  gripCyl.homeSensor[0]:= HomeSensor_gripCyl ;
  gripCyl.workSensor[0]:= WorkSensor_gripCyl ;
  HomeValve_gripCyl:= gripCyl.homeValve ;
  WorkValve_gripCyl:= gripCyl.workValve ;
  gripCyl.homeSensorLabel[0] := HomeLabel_gripCyl;
  gripCyl.workSensorLabel[0] := WorkLabel_gripCyl;
  
  jackCyl.homeSensor[0]:= HomeSensor_jackCyl ;
  jackCyl.workSensor[0]:= WorkSensor_jackCyl ;
  HomeValve_jackCyl:= jackCyl.homeValve ;
  WorkValve_jackCyl:= jackCyl.workValve ;
  jackCyl.homeSensorLabel[0] := HomeLabel_jackCyl;
  jackCyl.workSensorLabel[0] := WorkLabel_jackCyl;
  
  HomeValve_blow:= blow.homeValve ;
  WorkValve_blow:= blow.workValve ;
  
  fixCyl.homeSensor[0]:= HomeSensor_fixCyl ;
  fixCyl.workSensor[0]:= WorkSensor_fixCyl ;
  HomeValve_fixCyl:= fixCyl.homeValve ;
  WorkValve_fixCyl:= fixCyl.workValve ;
  fixCyl.homeSensorLabel[0] := HomeLabel_fixCyl;
  fixCyl.workSensorLabel[0] := WorkLabel_fixCyl;
  
  stepFixCyl.homeSensor[0]:= HomeSensor_stepFixCyl ;
  stepFixCyl.workSensor[0]:= WorkSensor_stepFixCyl ;
  HomeValve_stepFixCyl:= stepFixCyl.homeValve ;
  WorkValve_stepFixCyl:= stepFixCyl.workValve ;
  stepFixCyl.homeSensorLabel[0] := HomeLabel_stepFixCyl;
  stepFixCyl.workSensorLabel[0] := WorkLabel_stepFixCyl;
  
// Parameter 

  JacketStrippingData.Blow.homeSensorDisabled[0] := TRUE;
  JacketStrippingData.Blow.workSensorDisabled[0] := TRUE;
  
  rotateAxis.modulo.divisor := 2;
  rotateAxis.modulo.stepPoint :=1;
  rotateAxis.modulo.factor :=360;
  rotateAxis.modulo.mode := 1;
  rotateAxis.modulo.enable :=TRUE;
  rotateAxis.posUnit			:='deg';
  rotateAxis.veloUnit			:='deg/s';
  rotateAxis.accDecUnit	  :="deg/s²";
  
  cutAxis.movePosNum := 18;
  transferAxis.movePosNum := 15;
  rotateAxis.velocity :=1000;
  
  rotateAxis.Override := JacketStrippingData.CPP.override;
  TransferAxis.Override := JacketStrippingData.CPP.override;
  CutAxis.Override := JacketStrippingData.CPP.override;
  
  tonOn(IN:= onePlus, PT:= T#2S, Q=> , ET=> );
  tonOff(IN:= NOT onePlus, PT:= T#2S, Q=> , ET=> );
  IF tonOn.Q OR tonOff.Q THEN
    onePlus := NOT onePlus;
  END_IF
  
  mcWriteParameterPersistent(
    Axis:= rotateAxis.axis, 
    Execute:= onePlus, 
    ParameterNumber:= 1045, 
    Value:= 360.0, 
    Done=> , 
    Busy=> , 
    Error=> , 
    ErrorID=> );
    


//DATA 模拟

  IF NOT activated THEN
  
  activated:=TRUE;
  
  JacketStripping.Imm.Machine_airOn := TRUE;
  JacketStripping.Imm.Machine_allDoorClosed:= TRUE;
  JacketStripping.Imm.Machine_eStop:= TRUE;
  JacketStripping.Imm.Machine_safety:= TRUE;
  JacketStripping.Imm.Machine_manualMode:= TRUE;
  
  JacketStripping.Imm.carrierInPos := TRUE;
  JacketStripping.Imm.carrierPos := ENUM_CarrierPos.Left;
  JacketStripping.Imm.StationCanRun := TRUE;
  JacketStrippingData.CPP.override := 100;
  
  JacketStrippingData.CutAxis.movePos[HOME_CUT] := 40;
  JacketStrippingData.CutAxis.movePos[FIRST_PRECUT_CUT] := 30;
  JacketStrippingData.CutAxis.movePos[FIRST_CUT_CUT] := 10;
  JacketStrippingData.CutAxis.movePos[FIRST_BACK_CUT] := 20;
  JacketStrippingData.CutAxis.movePos[SECOND_PRECUT_CUT] := 25;
  JacketStrippingData.CutAxis.movePos[SECOND_CUT_CUT] :=5;
  JacketStrippingData.CutAxis.movePos[SECOND_BACK_CUT] := 15;
  
  JacketStrippingData.TransferAxis.movePos[HOME_TRANS] := 0;
  JacketStrippingData.TransferAxis.movePos[FIRST_CUT_TRANS] := 200;
  JacketStrippingData.TransferAxis.movePos[FIRST_BACK_TRANS] := 50;
  JacketStrippingData.TransferAxis.movePos[SECOND_CUT_TRANS] := 100;
  JacketStrippingData.TransferAxis.movePos[SECOND_BACK_TRANS] := 25;
  
  JacketStrippingData.GripCyl.homeSensorDisabled[0] := TRUE;
  JacketStrippingData.GripCyl.workSensorDisabled[0] := TRUE;
  JacketStrippingData.JackCyl.homeSensorDisabled[0] := TRUE;
  JacketStrippingData.JackCyl.workSensorDisabled[0] := TRUE;
  JacketStrippingData.FixCyl.homeSensorDisabled[0] := TRUE;
  JacketStrippingData.FixCyl.workSensorDisabled[0] := TRUE;
  JacketStrippingData.StepFixCyl.homeSensorDisabled[0] := TRUE;
  JacketStrippingData.StepFixCyl.workSensorDisabled[0] := TRUE;
  JacketStrippingData.GripCyl.homeTime := 500;
  JacketStrippingData.GripCyl.workTime := 500;
  JacketStrippingData.JackCyl.homeTime := 500;
  JacketStrippingData.JackCyl.workTime := 500;
  JacketStrippingData.FixCyl.homeTime := 500;
  JacketStrippingData.FixCyl.workTime := 500;
  JacketStrippingData.StepFixCyl.homeTime := 500;
  JacketStrippingData.StepFixCyl.workTime := 500;
  JacketStrippingData.Blow.homeTime := 500;
  JacketStrippingData.Blow.workTime := 500;
  
  END_IF
END_ACTION

ACTION StepAuto:
IF NOT station.initDone THEN
	station.flow[AUTO].actStep:=0;
ELSIF station.running 
THEN

CASE station.flow[AUTO].actStep OF

//	Home Step
0:
IF station.disabled
	AND station.canRun
  AND JacketStripping.Imm.allObjectInitPos
  AND NOT machine.stopping
  AND NOT station.cycleRunning
THEN
	JacketStripping.Imm.stationDone:=TRUE;
END_IF

IF (station.cycleRunning
		OR station.canRun
      AND JacketStripping.Imm.allObjectInitPos
			AND NOT station.Done
			AND NOT station.Disabled
      AND NOT machine.stopping
	)
	AND JacketStripping.Imm.carrierInPos
THEN
	station.flow[AUTO].actStep:=10;
	station.cycleTimeStart:=TRUE;
	station.cycleTimeEnd:=FALSE;
END_IF


//	fixCyl up
10:
IF JacketStripping.Imm.carrierPos= ENUM_CarrierPos.Left THEN
  fixCyl.auto:= TRUE;
  JacketStripping.Imm.carrierLeftProductState := 0;
	IF fixCyl.inWork THEN
		station.flow[AUTO].actStep:=station.flow[AUTO].actStep + 10;
	END_IF
ELSIF JacketStripping.Imm.carrierPos= ENUM_CarrierPos.Right THEN
  stepFixCyl.auto:= TRUE;
  JacketStripping.Imm.carrierRightProductState := 0;
	IF stepFixCyl.inWork THEN
		station.flow[AUTO].actStep:=station.flow[AUTO].actStep + 10;
	END_IF
END_IF


//	jackCyl up
20:
jackCyl.auto:=TRUE;
IF jackCyl.inWork THEN
	station.flow[AUTO].actStep:=station.flow[AUTO].actStep + 10;
END_IF

//	gripCyl close
30:
gripCyl.auto:=TRUE;
IF gripCyl.inWork THEN
	station.flow[AUTO].actStep:=station.flow[AUTO].actStep + 10;
END_IF

//transferAxis to firstCut pos
40:
transferAxis.moveAutoNo:=FIRST_CUT_TRANS;
IF transferAxis.inPos[FIRST_CUT_TRANS] THEN 
	station.flow[AUTO].actStep:=station.flow[AUTO].actStep + 10;
END_IF


//cutAxis to firstPreCut pos
50:
cutAxis.moveAutoNo:=FIRST_PRECUT_CUT;
rotateAxis.velocityAuto:=TRUE;
IF cutAxis.inPos[FIRST_PRECUT_CUT] THEN 
	station.flow[AUTO].actStep:=station.flow[AUTO].actStep + 10;
END_IF


//rotateAxis start
60:
IF rotateAxis.InVelocity THEN 
	station.flow[AUTO].actStep:=station.flow[AUTO].actStep + 10;
END_IF


//cutAxis to firstCut pos
70:
cutAxis.moveAutoNo:= FIRST_CUT_CUT;
IF cutAxis.inPos[FIRST_CUT_CUT] THEN 
	station.flow[AUTO].actStep:=station.flow[AUTO].actStep + 10;
END_IF
firstCutTimer(IN:=FALSE,PT:=UDINT_TO_TIME(JacketStrippingData.CPP.FirstCutTime),Q=>,ET=>);


//Wait firstCut delay
80:
firstCutTimer(IN:=TRUE,PT:=UDINT_TO_TIME(JacketStrippingData.CPP.FirstCutTime),Q=>,ET=>);
IF firstCutTimer.Q THEN
	station.flow[AUTO].actStep:=station.flow[AUTO].actStep + 10;
END_IF


//rotateAxis end
90:
  rotateAxis.stopAuto:=TRUE;
  IF rotateAxis.Axis.Status.NotMoving THEN
    rotateAxis.stopAuto:=FALSE;
    station.flow[AUTO].actStep:=station.flow[AUTO].actStep + 5;
	END_IF
  
//cutAxis to firstBack pos  
95:
  rotateAxis.stopAuto:=FALSE;
cutAxis.moveAutoNo:= FIRST_BACK_CUT;
IF cutAxis.inPos[FIRST_BACK_CUT] THEN 	
	station.flow[AUTO].actStep:=station.flow[AUTO].actStep + 5;
END_IF
firstOpenTimer(IN:=FALSE,PT:= UDINT_TO_TIME(JacketStrippingData.CPP.firstOpenTime),Q=>,ET=>);


//Wait firstOpen delay
100:
firstOpenTimer(IN:=TRUE,PT:=UDINT_TO_TIME(JacketStrippingData.CPP.firstOpenTime),Q=>,ET=>);
IF firstOpenTimer.Q THEN
	station.flow[AUTO].actStep:=station.flow[AUTO].actStep + 10;
END_IF

110:
//transferAxis to firstBack pos
transferAxis.moveAutoNo:=FIRST_BACK_TRANS;
IF transferAxis.inPos[FIRST_BACK_TRANS] THEN
	IF NOT JacketStrippingData.CPP.secondCutEnable THEN
		IF JacketStripping.Imm.carrierPos = ENUM_CarrierPos.Left THEN
			JacketStripping.Imm.carrierLeftProductState:=ENUM_ProductState.Good;
		ELSIF JacketStripping.Imm.carrierPos =ENUM_CarrierPos.Right THEN
			JacketStripping.Imm.carrierRightProductState:=ENUM_ProductState.Good;
		END_IF
		station.flow[AUTO].actStep:=900;
	ELSE
		station.flow[AUTO].actStep:=station.flow[AUTO].actStep + 10;
	END_IF
END_IF


//cutAxis to home pos
120:
cutAxis.moveAutoNo:= HOME_CUT;
IF cutAxis.inPos[HOME_CUT] THEN 
	station.flow[AUTO].actStep:=station.flow[AUTO].actStep + 80;
END_IF

//transferAxis to secondCut pos
200:
transferAxis.moveAutoNo:=SECOND_CUT_TRANS;
IF transferAxis.inPos[SECOND_CUT_TRANS] THEN
  	station.flow[AUTO].actStep:=station.flow[AUTO].actStep + 10;
END_IF


//cutAxis to secondPreCut pos
210:
rotateAxis.VelocityAuto:=TRUE;
cutAxis.moveAutoNo:= SECOND_PRECUT_CUT;
IF cutAxis.inPos[SECOND_PRECUT_CUT] THEN 
	station.flow[AUTO].actStep:=station.flow[AUTO].actStep + 10;
END_IF


//rotateAxis start
220:
IF rotateAxis.InVelocity THEN 
	station.flow[AUTO].actStep:=station.flow[AUTO].actStep + 10;
END_IF


//cutAxis to secondCut pos
230:

cutAxis.moveAutoNo:= SECOND_CUT_CUT;
IF cutAxis.inPos[SECOND_CUT_CUT] THEN 
	station.flow[AUTO].actStep:=station.flow[AUTO].actStep + 10;
END_IF
SecondCutTimer(IN:=FALSE,PT:=UDINT_TO_TIME(JacketStrippingData.CPP.SecondCutTime),Q=>,ET=>);


//Wait secondCut delay
240:
SecondCutTimer(IN:=TRUE,PT:=UDINT_TO_TIME(JacketStrippingData.CPP.SecondCutTime),Q=>,ET=>);
IF SecondCutTimer.Q THEN
	station.flow[AUTO].actStep:=station.flow[AUTO].actStep + 10;
END_IF

//rotateAxis end
250:
  rotateAxis.stopAuto:=TRUE;
  IF rotateAxis.Axis.Status.NotMoving THEN
    rotateAxis.stopAuto:=FALSE;
    station.flow[AUTO].actStep:=station.flow[AUTO].actStep + 5;
	END_IF
  
//cutAxis to firstBack pos  
255:
  rotateAxis.stopAuto:=FALSE;
cutAxis.moveAutoNo:= SECOND_BACK_CUT;
IF cutAxis.inPos[SECOND_BACK_CUT] THEN 	
	station.flow[AUTO].actStep:=station.flow[AUTO].actStep + 5;
END_IF
secondOpenTimer(IN:=FALSE,PT:=UDINT_TO_TIME(JacketStrippingData.CPP.secondOpenTime),Q=>,ET=>);


//Wait secondOpen delay
260:
secondOpenTimer(IN:=TRUE,PT:=UDINT_TO_TIME(JacketStrippingData.CPP.secondOpenTime),Q=>,ET=>);
IF secondOpenTimer.Q THEN
	station.flow[AUTO].actStep:=station.flow[AUTO].actStep + 10;
END_IF


//transferAxis to secondBack pos
270:
transferAxis.moveAutoNo:=SECOND_BACK_TRANS;
IF transferAxis.InPos[SECOND_BACK_TRANS] THEN
	IF JacketStripping.Imm.carrierPos = ENUM_CarrierPos.Left THEN
		JacketStripping.Imm.carrierLeftProductState:=ENUM_ProductState.Good;
	ELSIF JacketStripping.Imm.carrierPos = ENUM_CarrierPos.Right THEN
		JacketStripping.Imm.carrierLeftProductState:=ENUM_ProductState.Good;
	END_IF
	station.flow[AUTO].actStep:=station.flow[AUTO].actStep + 30;
END_IF


//cutAxis to home pos
900:
cutAxis.moveAutoNo := HOME_CUT;
IF cutAxis.InPos[HOME_CUT] THEN 
	station.flow[AUTO].actStep:=station.flow[AUTO].actStep + 10;
END_IF


//transferAxis&rotateAxis to home pos
910:
transferAxis.moveAutoNo:= HOME_TRANS;
rotateAxis.moveAutoNo:=HOME_ROTATE;
IF transferAxis.InPos[HOME_TRANS]
	AND rotateAxis.inPos[HOME_ROTATE]
THEN 
	station.flow[AUTO].actStep:=station.flow[AUTO].actStep + 10;
END_IF


//gripCyl home
920:
gripCyl.auto:=FALSE;
IF gripCyl.inHome THEN
	station.flow[AUTO].actStep:=station.flow[AUTO].actStep + 10;
END_IF


//fixCyl jackCyl home
930:
fixCyl.auto:=FALSE;
stepFixCyl.auto:=FALSE;
jackCyl.auto:=FALSE;
IF fixCyl.inHome
	AND jackCyl.inHome
	AND stepFixCyl.inHome
THEN
	station.flow[AUTO].actStep:=999;
END_IF
blowTimer(IN:=FALSE,PT:=UDINT_TO_TIME(JacketStrippingData.CPP.blowTime),Q=>,ET=>);

//blow start
940:
blow.auto:=TRUE;
blowTimer(IN:=TRUE,PT:=UDINT_TO_TIME(JacketStrippingData.CPP.blowTime),Q=>,ET=>);
IF blowTimer.Q THEN
	station.flow[AUTO].actStep:=station.flow[AUTO].actStep + 10;
END_IF


//blow stop
950:
blow.Auto:=FALSE;
station.flow[AUTO].actStep:=999;


//	Single Run Finish
999:
station.cycleRunFlag:=FALSE;
station.flow[AUTO].actStep:=0;
station.cycleTimeStart:=FALSE;
station.cycleTimeEnd:=TRUE;
JacketStripping.Imm.stationDone:=TRUE;
END_CASE

END_IF
END_ACTION

ACTION StepInit:
IF NOT station.Initing THEN
	station.flow[INIT].actStep:=0;
ELSE

CASE station.flow[INIT].actStep OF
//	Home Step
0:
IF station.Initing
	AND NOT station.InitDone
THEN
	station.flow[INIT].actStep:=station.flow[INIT].actStep + 10;
END_IF

//	Axis Power
10:
rotateAxis.stopAuto:=TRUE;
rotateAxis.VelocityAuto:=FALSE;
cutAxis.PowerInit:=TRUE;
rotateAxis.PowerInit:=TRUE;
transferAxis.PowerInit:=TRUE;
IF rotateAxis.isPowerOn
	AND transferAxis.isPowerOn
	AND cutAxis.isPowerOn
THEN
station.flow[INIT].actStep:=station.flow[INIT].actStep + 10;
END_IF

//	cutAxis home
20:
rotateAxis.stopAuto:=FALSE;
cutAxis.moveAutoNo :=HOME_CUT;
IF cutAxis.inPos[HOME_CUT] THEN
  station.flow[INIT].actStep:=station.flow[INIT].actStep + 10;
END_IF

//	transferAxis home
30:
transferAxis.moveAutoNo:= HOME_TRANS;
IF transferAxis.inPos[HOME_TRANS] THEN
  station.flow[INIT].actStep:=station.flow[INIT].actStep + 10;
END_IF

//	gripCyl home
40:
gripCyl.homeInit:=TRUE;
IF gripCyl.inHome THEN
	station.flow[INIT].actStep:=station.flow[INIT].actStep + 10;
END_IF


//	fixCyl down
50:
jackCyl.homeInit:=TRUE;
fixCyl.homeInit:=TRUE;
stepFixCyl.homeInit:=TRUE;
blow.homeInit:=TRUE;
IF fixCyl.inHome 
	AND stepFixCyl.inHome
	AND jackCyl.inHome
  AND blow.inHome
THEN
	station.flow[INIT].actStep:=station.flow[INIT].actStep + 10;
END_IF


//	rotateAixs home
60:
rotateAxis.moveAutoNo:= HOME_ROTATE;
IF rotateAxis.inPos[HOME_ROTATE] THEN
	station.flow[INIT].actStep:=999;
END_IF


//	Init Done
999:
station.flow[INIT].actStep:=0;
station.InitDone:=1;

END_CASE

END_IF
END_ACTION

ACTION Tip:

END_ACTION

END_FUNCTION_BLOCK

// ---- Standard/Public/02 Station/FB_Station_RD.TcPOU
FUNCTION_BLOCK FB_Station_RD
VAR_INPUT
END_VAR
VAR_OUTPUT
END_VAR
VAR_IN_OUT
machine : UDT_Machine_RD; //
station : UDT_Station_RD; //  

END_VAR

VAR
END_VAR

VAR
safetyPermit : BOOL; // 安全条件
stationIniting : Bool; // 单工站初始化中
singleRunFlagCache : Bool; // 单循环标志缓存
machineInit : Bool; // 整机初始化执行
initExecute : Bool; // 初始化执行
cycleRunExecute : Bool; // 单循环执行
jogRunExecute : Bool; // 寸动执行
initingCache : Bool; // 整机初始化缓存
inithmiCache : Bool; // 初始化hmi缓存
initAutoCache : Bool; // 初始化AutoI缓存
cycleRunhmiCache : Bool; // 单循环hmi缓存
cycleRunAutoCache : Bool; // 单循环AutoI缓存
jogRunhmiCache : Bool; // 寸动hmi下缓存
cycleTimeEndCache : Bool; // 工站周期结束缓存
cycleTimeTimer : TON; // 工站周期定时器
initingTimer : TON; // 初始化中定时器
initTimeoutTimer : TON; // 初始化超时定时器
jogRunhmiTimer : TON; // 寸动按下定时器
isJogRunhmiTimer : BOOL; //寸动按下定时到位
isInitTimeoutTimer : BOOL; //
flowNum : UINT; // 流程数量
flowTimeoutTimer : ARRAY[0..5] OF TON ; // 流程步超时定时器
isFlowTimeout : Array[0..5] of BOOL; //
flowStepCache : Array[0..5] of UInt; // 流程步缓存
language : INT; //
index : UINT; //
activated : Bool; //

END_VAR

VAR CONSTANT
MAX_FLOW : UINT:=5; // 流程最大数量

STATE_ALARM : UInt:=0; // 报警中
STATE_NOT_READY : UInt:=1; // 未准备就绪
STATE_READY : UInt:=2; // 准备就绪
STATE_RUNNING : UInt:=3; // 运行中
STATE_SINGLE_RUN : UInt:=4; // 单循环中
STATE_SINGLE_PAUSE : UInt:=5; // 单循环暂停
STATE_INITING : UInt:=6; // 初始化中
STATE_NOT_INIT : UINT:=7; // 未初始化

INIT_TIMEOUT : UInt:=1; // 初始化超时报警
NOT_INIT_NOT_START : UInt:=2; // 未初始化不能启动
SINGLE_RUN_NOT_START : UInt:=3; // 单循环中不能启动
FLOW_TIMEOUT : UInt:=4; // 流程超时
NOT_RUN_PERMIT : UInt:=5; // 工站运行条件不足
AUTO_TIP_POPUP : UINT:=11; //  自动提示弹窗
END_VAR

SetUp();
Flow();
Alarm();
AutoTip();
ManualTip();
General();
Init();
Running();
Status();
CycleTime();

ACTION Alarm:
//-----------------------------------Alarm-----------------------------------------//
  
  IF isInitTimeoutTimer  THEN
    station.presetAlarms[0] := TRUE;//工站初始化超时报警
  END_IF;
    
  //工站报警中 
  station.alarming :=
  FUN_AryBitCount_RD(station.presetAlarms) >0 
  OR FUN_AryBitCount_RD(station.userAlarms) >0 
  OR station.report.alarming ;
   
  IF FUN_AryBitCount_RD(station.presetAlarms) >0 THEN
    machine.alarmCount :=machine.alarmCount + FUN_AryBitCount_RD(station.presetAlarms);
  END_IF;
  IF FUN_AryBitCount_RD(station.userAlarms) >0 THEN
    machine.alarmCount :=machine.alarmCount  + FUN_AryBitCount_RD(station.userAlarms);
  END_IF;
  
  //反馈机器报警
  IF station.alarming THEN
    station.running := FALSE;
    station.initing := FALSE;
    machine.report.stationAlarming := TRUE;
  END_IF;
  
  //报警复位
  IF machine.reset THEN
    MEMSET(destAddr:=ADR(station.presetAlarms) , fillByte:= 0, n:=SIZEOF(station.presetAlarms));
    MEMSET(destAddr:=ADR(station.userAlarms) , fillByte:= 0, n:=SIZEOF(station.userAlarms));

    station.report.alarming := FALSE;   //复位下级报警
  END_IF;
  
//-----------------------------------------------------------------------------------//*)
END_ACTION

ACTION AutoTip:
//-----------------------------------AutoTip-----------------------------------------//
  
  //工站未初始化
  station.presetAutoTips[0] := NOT station.initDone;
  //工站单循环中
  station.presetAutoTips[1] := machine.autoMode AND station.cycleRunFlag;
  //工站运行条件不足
  station.presetAutoTips[2] := NOT station.runPermit;
  
  //工站自动提示
  station.autoTip :=
  FUN_AryBitCount_RD(station.presetAutoTips) >0 
  OR FUN_AryBitCount_RD(station.userAutoTips) >0 
  OR station.report.autoTip;
  station.report.autoTip := FALSE;
  
  //自动提示弹窗
  IF station.autoTip AND (station.cycleRunhmi OR station.jogRunhmi) THEN
    station.autoTipTrigger := TRUE;
    machine.popup := AUTO_TIP_POPUP;
  END_IF;
  IF machine.popup = 0 THEN
    station.autoTipTrigger := FALSE;
  END_IF;

  //反馈机器自动提示
  IF station.autoTip THEN
    machine.report.stationAutoTip := TRUE;
  END_IF;
  
//-----------------------------------------------------------------------------------//*)
END_ACTION

ACTION CycleTime:
//-----------------------------------CycleTime-------------------------------------//
  //工站周期计时
  IF cycleTimeEndCache THEN
    station.cycleTimeEnd := FALSE;
  ELSIF station.cycleTimeEnd THEN
    station.cycleTime := TIME_TO_DINT (cycleTimeTimer.ET);
    station.cycleTimeStart := FALSE;
  END_IF;
  cycleTimeTimer(IN := station.cycleTimeStart,
                  //Reset := (NOT cycleTimeEndCache AND station.cycleTimeEnd) // 工站周期结束上升沿
                  //OR station.initing,
                  PT := T#1000S,
  );
  cycleTimeEndCache := station.cycleTimeEnd;
  
//-----------------------------------------------------------------------------------//*)
END_ACTION

ACTION Flow:
//-----------------------------------Flow-----------------------------------------//
station.flowDisplay:= LINT_TO_UINT( MIN(station.flowDisplay,SIZEOF(machine.flow) -1));
flowNum := station.flowDisplay;
  //流程监控
  FOR index := 0 TO flowNum DO
    IF station.flow[index].actStep = 999 THEN
      station.flow[index].uninterrupted := TRUE;
    END_IF;
    //流程上一步记录
    IF station.flow[index].actStep <> flowStepCache[index] THEN
      station.flow[index].prevStep := flowStepCache[index];
    END_IF;
    flowStepCache[index] := station.flow[index].actStep;
    //流程超时计时
    flowTimeoutTimer[index](IN := station.flow[index].timeoutEnable
			AND NOT station.flow[index].timeoutException
			AND NOT station.disabled
			AND (station.running OR station.initing)
			AND station.flow[index].actStep > 0
			AND station.flow[index].actStep = flowStepCache[index],     
			PT := station.flow[index].setTimeout,
			Q=>isFlowTimeout[index]);
    station.flow[index].timeoutException := FALSE;
    //流程超时报警置位
    IF isFlowTimeout[index] THEN
      station.flow[index].timeoutAlarm := TRUE;
      station.presetAlarms[index + 8] := TRUE;
    ELSIF machine.reset THEN
      station.flow[index].timeoutAlarm := FALSE;
    END_IF;
  END_FOR;
//-----------------------------------------------------------------------------------//*)
END_ACTION

ACTION General:
//-----------------------------------General----------------------------------------//
  
  //安全条件
  safetyPermit := machine.eStop
  AND machine.airOn
  AND machine.safety
  AND machine.allDoorClosed;
  
  //准备就绪
  station.ready := safetyPermit
  AND station.initDone
  AND station.runPermit
  AND NOT machine.publicAlarm
  AND NOT station.alarming
  AND NOT station.autoTip;
  
  // 初始化允许操作
  station.initAllow :=safetyPermit
  AND station.initPermit
  AND NOT machine.publicAlarm
  AND NOT station.alarming;
  // 单循环允许操作
  station.cycleRunAllow := station.ready AND station.cycleRunPermit;
  // 寸动允许操作
  station.jogRunAllow := station.ready AND station.jogRunPermit;
  // 禁止图标
  station.initForbidIcon := NOT station.initAllow OR NOT machine.manualMode;
  station.cycleRunForbidIcon := NOT station.cycleRunAllow OR NOT machine.manualMode;
  station.jogRunForbidIcon := NOT station.jogRunAllow OR NOT machine.manualMode;
  
//-----------------------------------------------------------------------------------//*)
END_ACTION

ACTION Init:
//-----------------------------------Init-----------------------------------------//
  // 单工站初始化执行
  initExecute :=
  inithmiCache AND NOT station.inithmi // inithmi下降沿
  OR NOT initAutoCache AND station.initAuto // initAuto上升沿
  OR station.initSyncMachine AND NOT initingCache AND machine.initing; // 整机初始化上升沿
  inithmiCache := station.inithmi;
  initAutoCache := station.initAuto;
  initingCache := machine.initing;
  station.initAuto := FALSE;
  // 启用急停后需初始化或初始化时先复位初始化完成
  IF (NOT machine.eStop AND station.requiresReinitialize) // 急停
    OR (initExecute AND station.initAllow)  // 初始化执行
  THEN
    station.initDone := FALSE;
    station.cycleRunFlag := FALSE;
    station.cycleTimeStart := FALSE;
    station.cycleTimeEnd := FALSE;
    station.flow[0].nextStep := 0;
    station.flow[0].actStep := 0;
    station.flow[0].prevStep := 0;
  END_IF;
  //单工站初始化中
  IF station.initAllow
    AND NOT station.initDone
    AND NOT station.pausehmi
    AND NOT machine.pause
  THEN
    IF initExecute AND station.initAllow THEN
      stationIniting := TRUE;
    END_IF;
  ELSE
    stationIniting := FALSE;
  END_IF;
  //工站初始化中
  station.initing := stationIniting;
  //初始化延时
	initingTimer(IN := station.initing,
				PT := T#10S,
				Q => station.initDelay);
  
  //初始化复位自动流程
  IF station.initResetAutoFlow
    AND station.initing
    AND NOT station.initDelay
  THEN
    FOR index := 1 TO MAX_FLOW DO
      station.flow[index].nextStep := 0;
      station.flow[index].actStep := 0;
      station.flow[index].prevStep := 0;
    END_FOR;
  END_IF;
  //初始化超时
	initTimeoutTimer(IN := station.initing,
				PT := station.initTimeout,
				Q=>isInitTimeoutTimer
	);
  //反馈给机器初始化未完成
  IF NOT station.initDone THEN
    machine.report.stationNotInitDone := TRUE;
  END_IF;
//-----------------------------------------------------------------------------------//
END_ACTION

ACTION ManualTip:
//-----------------------------------ManualTip-----------------------------------------//
  
  //复位手动提示    
  IF machine.tipReset THEN
   MEMSET(destAddr:=ADR(station.presetManualTips) , fillByte:= 0, n:=SIZEOF(station.presetManualTips));
   MEMSET(destAddr:=ADR(station.userManualTips) , fillByte:= 0, n:=SIZEOF(station.userManualTips));
  END_IF;
  
  //手动提示
  IF station.cycleRunhmi OR station.jogRunhmi OR station.inithmi THEN
    machine.presetManualTips[0] := NOT machine.eStop;     //急停中,无法操作
    machine.presetManualTips[1] := NOT machine.safety;    //安全条件不满足,无法操作
    machine.presetManualTips[2] := NOT machine.allDoorClosed;  //安全门未锁好,无法操作
    machine.presetManualTips[3] := NOT machine.airOn;     //气压不足,无法操作
    machine.presetManualTips[4] := NOT machine.manualMode;//不在手动模式,无法操作
  END_IF;
  
  //手动提示中
  station.manualTip :=
  FUN_AryBitCount_RD(station.presetManualTips) >0 
  OR FUN_AryBitCount_RD(station.userManualTips) >0 
  OR station.report.manualTip;
  
  //反馈整机手动提示
  IF station.manualTip THEN
    machine.report.stationManualTip := TRUE;
  END_IF;
  
//-----------------------------------------------------------------------------------//
END_ACTION

ACTION Running:
//-----------------------------------Running---------------------------------------//
  
  // 单循环执行
  cycleRunExecute := cycleRunhmiCache AND NOT station.cycleRunhmi
  OR NOT cycleRunAutoCache AND  station.cycleRunAuto;
  cycleRunhmiCache := station.cycleRunhmi;
  cycleRunAutoCache :=  station.cycleRunAuto;
  station.cycleRunAuto := FALSE;
  // 寸动执行
  jogRunExecute := jogRunhmiCache AND NOT station.jogRunhmi;
  jogRunhmiCache := station.jogRunhmi;
  jogRunhmiTimer(IN := station.jogRunhmi,
	          PT := T#1S,
			  Q=>isJogRunhmiTimer
		  );
  IF machine.eStop AND station.initDone THEN
    IF (cycleRunExecute AND station.cycleRunAllow
      OR jogRunExecute AND station.jogRunAllow)
      AND station.ready
      AND machine.manualMode
    THEN
      station.cycleRunFlag := TRUE;
    END_IF;
    // 单循环标志下降沿 and 单循环重复功能开启
    IF singleRunFlagCache AND NOT station.cycleRunFlag
      AND station.repetitionsEnable
    THEN
      station.repetitions := station.repetitions +1;  //单循环次数加1
      // 单循环计次<设定次数
      station.cycleRunFlag := station.repetitions < station.repetitionsTimes;
    END_IF;
  ELSE
    station.cycleRunFlag := FALSE;
  END_IF;
  singleRunFlagCache := station.cycleRunFlag;
  // 单循环中、寸动中
  IF station.ready
    AND machine.manualMode
    AND station.cycleRunFlag
    AND NOT station.pausehmi
    AND NOT machine.pause
  THEN
    IF cycleRunExecute AND station.cycleRunAllow THEN
      station.cycleRunning := TRUE;
    END_IF;
    station.jogRunning := jogRunExecute AND station.jogRunAllow     //按下去一秒钟内，点一次动一次
    OR isJogRunhmiTimer;   //按下去超过一秒钟后，点着动，松开停
  ELSE
    station.cycleRunning := FALSE;
    station.jogRunning := FALSE;
  END_IF;
  
  // 运行中
  IF machine.manualMode THEN
    station.running := station.cycleRunning OR station.jogRunning; // 手动模式下工站单循环和工站寸动
  ELSIF machine.autoMode OR machine.jogMode THEN  // 自动模式下整机运行或整机寸动
    IF station.ready
      AND NOT machine.paused
      AND NOT machine.stopDone
    THEN
      IF machine.running THEN
        station.running := TRUE;
      ELSIF station.syncAlarms THEN
        station.running := FALSE;
      END_IF;
    ELSE
      station.running := FALSE;
    END_IF;
  ELSE
    station.running := FALSE;
  END_IF;
  
//-----------------------------------------------------------------------------------//
END_ACTION

ACTION SetUp:
//-----------------------------------SetUp-----------------------------------------//

  IF NOT activated THEN
	  activated:=TRUE;
	//赋初始值
	station.cycleRunPermit		:=TRUE;
	station.	jogRunPermit			:=TRUE;
	station.	disablePermit			:=TRUE;
	station.	requiresReinitialize	:=TRUE;
	station.initPermit			:=TRUE;
	station.runPermit			:=TRUE;
	station.canRun				:=TRUE;
	station.initTimeout		:=T#30s;
    //流程数量
	station.flowDisplay:=2;
	FOR index:=0 TO 5 DO
		station.flow[index].timeoutEnable	:=TRUE;
	    station.flow[index].setTimeout			:=T#30s;
	END_FOR;

  END_IF;
//-----------------------------------------------------------------------------------//
END_ACTION

ACTION Status:
//-----------------------------------Status
  
  IF station.alarming THEN
    station.status := STATE_ALARM;
  ELSIF station.initing THEN
    station.status := STATE_INITING;
  ELSIF NOT station.initDone THEN
    station.status := STATE_NOT_INIT;
  ELSIF NOT station.ready THEN
    station.status := STATE_NOT_READY;
  ELSIF station.cycleRunning THEN
    station.status := STATE_SINGLE_RUN;
  ELSIF station.cycleRunFlag THEN
    station.status := STATE_SINGLE_PAUSE;
  ELSIF station.running THEN
    station.status := STATE_RUNNING;
  ELSE
    station.status := STATE_READY;
  END_IF;
  
//-----------------------------------------------------------------------------------//
END_ACTION

END_FUNCTION_BLOCK

// ---- Standard/FUN/FUN_AryBitCount_RD.TcPOU
FUNCTION FUN_AryBitCount_RD : UINT
VAR_IN_OUT
 IN : ARRAY[*] OF BOOL;
END_VAR
VAR  
  index : INT;
END_VAR

FUN_AryBitCount_RD:=0;
FOR index:=0 TO SIZEOF(IN)-1 DO
	IF IN[index] THEN
    FUN_AryBitCount_RD := FUN_AryBitCount_RD +1 ;
	END_IF;	
END_FOR;

END_FUNCTION

// ---- Standard/Unit/05 Cylinder/FB_Cylinder_RD.TcPOU
FUNCTION_BLOCK FB_Cylinder_RD

VAR_INPUT
END_VAR

VAR_OUTPUT
END_VAR

VAR_IN_OUT
machine : UDT_Machine_RD; //
station : UDT_Station_RD; //
vari : UDT_CylinderVar_RD; //
data : UDT_CylinderData_RD; //
END_VAR

VAR
END_VAR

VAR
safetyPermit : BOOL; // 安全条件
sensorOn : Array[0..3] of Bool; // 感应器On时的正常状态，由气缸数量决定
sensorOff : Array[0..3] of Bool; // 感应器Off时的正常状态，由气缸数量决定
index : UINT; //
workValveCache : Bool; //
homeValveCache : Bool; //
workhmiCache : Bool; //
homehmiCache : Bool; //
resetCache : Bool; //
toWorkActionTimer : TON; // 去动点位置定时器
toHomeActionTimer : TON; // 去原点位置定时器
atWorkPosTimer : TON; // 在动点位置定时器
atHomePosTimer : TON; // 在原点位置定时器
alarmTimer : TON; // 报警定时器
isAlarmTime : BOOL; //FALSE
activated : BOOL; //FALSE
END_VAR

VAR CONSTANT
HOME_SENSOR_OFF_ALARM : UINT := 1; // 原点无信号报警  
WORK_SENSOR_OFF_ALARM : UINT := 2; // 动点无信号报警
HOME_SENSOR_ON_ALARM : UINT := 3; // 原点有信号报警
WORK_SENSOR_ON_ALARM : UINT := 4; // 动点有信号报警
IN_MANUAL : UINT := 5; // 气缸手动操作中
NO_HOME_PERMIT : UINT := 6; // 原点动作条件不满足
NO_WORK_PERMIT : UINT := 7; // 动点动作条件不满足
ALARM_TIME : UINT := 1; // 报警延时2，报警延时后，感应器异常延时
END_VAR

SetUp();
General();
Manual();
Init();
Output();
Delay();
Alarm();
ManualTip();
AutoTip();
Cache();

ACTION Alarm:
//----------------------------------Alarm-----------------------------------------//
  
  // 先复位报警，报警是优先于复位
  IF NOT resetCache AND machine.reset THEN
    vari.homeSensorOffAlarm := sensorOff;
    vari.workSensorOffAlarm := sensorOff;
    vari.homeSensorOnAlarm := sensorOff;
    vari.workSensorOnAlarm := sensorOff;
  END_IF;
  
  // 阀输出延时，有气压信号时才启动延时报警
  toHomeActionTimer(
                     IN := machine.airOn AND vari.homeValve,
                     PT := UDINT_TO_TIME(data.alarmTime+data.homeTime)//防止到位延时设置得比报警延时还长，导致的误报警
  );
  toWorkActionTimer(
                     IN := machine.airOn AND vari.workValve,
                     PT := UDINT_TO_TIME(data.alarmTime+data.workTime) //防止到位延时设置得比报警延时还长，导致的误报警
  );
  
  //  报警延时，用到位延时防止感应器抖动时无报警
  alarmTimer(IN := toHomeActionTimer.Q AND NOT vari.inHome
              OR toWorkActionTimer.Q AND NOT vari.inWork,
              PT := DINT_TO_TIME(ALARM_TIME),
			  Q=>isAlarmTime
  );

  // 报警输出
  IF isAlarmTime THEN
    FOR index := 0 TO vari.controlCylNum - 1 DO
      IF vari.homeValve THEN   //判断感应器与阀的状态不对应就置位报警字，且OR报警字进行保持
        vari.homeSensorOffAlarm[index] := vari.homeSensorOffAlarm[index] OR (vari.homeSensor[index] XOR sensorOn[index]);
        vari.workSensorOnAlarm[index] := vari.workSensorOnAlarm[index] OR (vari.workSensor[index] AND sensorOn[index]);
      ELSIF vari.workValve THEN
        vari.workSensorOffAlarm[index] := vari.workSensorOffAlarm[index] OR (vari.workSensor[index] XOR sensorOn[index]);
        vari.homeSensorOnAlarm[index] := vari.homeSensorOnAlarm[index] OR (vari.homeSensor[index] AND sensorOn[index]);
      END_IF;
    END_FOR;
  END_IF;
  
  // 气缸报警中
	FOR index := 0 TO vari.controlCylNum - 1 DO
		IF  vari.homeSensorOffAlarm[index] 
		    OR vari.workSensorOffAlarm[index] 
			OR vari.homeSensorOnAlarm[index] 
			OR vari.workSensorOnAlarm[index] 
		THEN
		  vari.alarming :=TRUE;
		  EXIT;
		ELSIF index= vari.controlCylNum - 1 THEN
			  vari.alarming :=FALSE;
	  	END_IF;
  	END_FOR;
  
  //反馈报警中
  IF vari.alarming THEN
    machine.alarmCount := machine.alarmCount + 1;
    station.report.alarming := TRUE;
  END_IF;
//-----------------------------------------------------------------------------------//
END_ACTION

ACTION AutoTip:
//----------------------------------AutoTip-----------------------------------------//
  
  //自动提示
  vari.autoTip := vari.manual;
  
  //反馈工站自动提示
  IF vari.autoTip THEN
    station.report.autoTip := TRUE;
  END_IF;
  
//-----------------------------------------------------------------------------------//
END_ACTION

ACTION Cache:
//----------------------------------Cache-----------------------------------------//
  
  resetCache := machine.reset;
  homehmiCache := vari.homehmi;
  workhmiCache := vari.workhmi;
  homeValveCache := vari.homeValve;
  workValveCache := vari.workValve;
  vari.homeInit := FALSE;
  vari.workInit := FALSE;
//-----------------------------------------------------------------------------------//
END_ACTION

ACTION Delay:
//----------------------------------Delay-------------------------------------------//
  //  原点延时
  IF vari.homeValve THEN
    vari.inWork := FALSE;
    atHomePosTimer(
                    IN := machine.airOn
                    AND vari.homeValve
                    AND NOT vari.workValve
                    AND vari.homeSensor[0] = sensorOn[0]     
					AND vari.homeSensor[1] = sensorOn[1]  
					AND vari.homeSensor[2] = sensorOn[2]  
					AND vari.homeSensor[3] = sensorOn[3]  //已配置的原点感应器ON
					AND NOT vari.workSensor[0]
					AND NOT vari.workSensor[1]
					AND NOT vari.workSensor[2]
                    AND NOT vari.workSensor[3],   //所有动点感应OFF
                    PT := UDINT_TO_TIME(data.homeTime),
                    Q => vari.inHome);
  ELSIF vari.workValve THEN
    // 动点延时
    vari.inHome := FALSE;
    atWorkPosTimer(
                    IN := machine.airOn
                    AND NOT vari.homeValve
                    AND vari.workValve
					AND NOT vari.homeSensor[0]  
					AND NOT vari.homeSensor[1]  
					AND NOT vari.homeSensor[2]  
                    AND NOT vari.homeSensor[3]   //所有原点感应OFF
                    AND vari.workSensor[0] = sensorOn[0],    //已配置的动点感应器ON
                    PT := UDINT_TO_TIME(data.workTime),
                    Q => vari.inWork);
  ELSE
    vari.inHome := FALSE;
    vari.inWork := FALSE;
  END_IF;

  //  气缸动作用时
  IF vari.busy THEN
    IF vari.inHome THEN
      vari.toHomeActionTime := TIME_TO_UDINT(toHomeActionTimer.ET);
    END_IF;
    IF vari.inWork THEN
      vari.toWorkActionTime := TIME_TO_UDINT(toWorkActionTimer.ET);
    END_IF;
  ELSIF NOT homeValveCache AND vari.homeValve THEN
    vari.toHomeActionTime := 0;
  ELSIF NOT workValveCache AND vari.workValve THEN
    vari.toWorkActionTime := 0;
  END_IF;
  
  // Busy信号，阀有输出且未到位对于点就是Busy
  vari.busy := NOT vari.alarming
  AND (vari.homeValve AND NOT vari.workValve AND NOT vari.inHome
  OR vari.workValve AND NOT vari.homeValve AND NOT vari.inWork);
  
//-----------------------------------------------------------------------------------//
END_ACTION

ACTION General:
//----------------------------------General-----------------------------------------//
  
  //安全条件
  safetyPermit := machine.eStop
  AND machine.safety
  AND machine.airOn
  AND machine.allDoorClosed;
  
  IF vari.controlCylNum > 0 THEN
    // 屏蔽气缸感应器时,感应器的状态直接与电磁阀输出关联
    FOR index := 0 TO vari.controlCylNum - 1 DO
      IF data.homeSensorDisabled[index] THEN
        vari.homeSensor[index] := vari.homeValve;
      END_IF;
      IF data.workSensorDisabled[index] THEN
        vari.workSensor[index] := vari.workValve;
      END_IF;
    END_FOR;
    	
  END_IF;
  
//-----------------------------------------------------------------------------------//
END_ACTION

ACTION Init:
//----------------------------------Init-----------------------------------------//
  
  IF safetyPermit THEN
    IF vari.homeInit THEN
      vari.enabled := TRUE;
      vari.manual := FALSE;
      vari.auto := FALSE;
    ELSIF vari.workInit THEN
      vari.enabled := TRUE;
      vari.manual := FALSE;
      vari.auto := TRUE;
    END_IF;
  ELSIF NOT machine.eStop AND vari.estoppedReInit THEN
    vari.enabled := FALSE;  //  当estoppedReInit :=true时急停会断开使能
  END_IF;
  
//-----------------------------------------------------------------------------------//
END_ACTION

ACTION Manual:
//----------------------------------Manual-----------------------------------------//
  
  IF safetyPermit AND machine.manualMode THEN
    vari.homeForbidIcon := NOT vari.homePermit;//原点禁止图标
    IF vari.homePermit AND homehmiCache AND NOT vari.homehmi THEN
      vari.manual := vari.auto;
      vari.enabled := TRUE;
    END_IF;
    vari.workForbidIcon := NOT vari.workPermit;//动点禁止图标
    IF vari.workPermit AND workhmiCache AND NOT vari.workhmi THEN
      vari.manual := NOT vari.auto;
      vari.enabled := TRUE;
    END_IF;
  ELSE
    vari.homeForbidIcon := TRUE;
    vari.workForbidIcon := TRUE;
  END_IF;
  
  vari.homeManual := vari.manual AND vari.auto;
  vari.workManual := vari.manual AND NOT vari.auto;
  
//-----------------------------------------------------------------------------------//
END_ACTION

ACTION ManualTip:
//----------------------------------ManualTip--------------------------------------//
  
  IF machine.tipReset THEN
    vari.noHomePermitManualTip := FALSE;
    vari.noWorkPermitManualTip := FALSE;
  ELSIF vari.homehmi OR vari.workhmi THEN
    machine.presetManualTips[0] := NOT machine.eStop;     //急停中,无法操作
    machine.presetManualTips[1] := NOT machine.safety;    //安全条件不满足,无法操作
    machine.presetManualTips[2] := NOT machine.allDoorClosed;  //安全门未锁好,无法操作
    machine.presetManualTips[3] := NOT machine.airOn;     //气压不足,无法操作
    machine.presetManualTips[4] := NOT machine.manualMode;//不在手动模式,无法操作
    
    IF safetyPermit AND machine.manualMode THEN
      IF NOT vari.homePermit AND vari.homehmi THEN
        vari.noHomePermitManualTip := TRUE;//原点条件不满足，用于置位外部提示信息用
      ELSIF NOT vari.workPermit AND vari.workhmi THEN
        vari.noWorkPermitManualTip := TRUE;//动点条件不满足，用于置位外部提示信息用
      END_IF;
    END_IF;
    
  END_IF;
  
  //反馈工站手动提示
  IF vari.noHomePermitManualTip
    OR vari.noWorkPermitManualTip
  THEN
    station.report.manualTip := TRUE;
  END_IF;
  
//-----------------------------------------------------------------------------------//
END_ACTION

ACTION Output:
//----------------------------------Output-----------------------------------------//
  
  //  原点阀输出
  vari.homeValve := vari.enabled
  AND NOT vari.release
  AND NOT (vari.manual XOR vari.auto);
  
  //  动点阀输出
  vari.workValve := vari.enabled
  AND NOT vari.release
  AND (vari.manual XOR vari.auto);
  
//-----------------------------------------------------------------------------------//
END_ACTION

ACTION SetUp:
//----------------------------------SetUp-----------------------------------------//
  
  IF NOT activated THEN
	activated:=TRUE;
	vari.homePermit:=TRUE;
	vari.workPermit:=TRUE;
	vari.controlCylNum:=1;
	vari.stationNo:=0;
	IF data.alarmTime = 0 THEN
		data.alarmTime :=5000;
	END_IF;
  END_IF;
    //根据气缸数，确定打开时传感器的状态,最大4个气缸
    vari.controlCylNum := LIMIT(UINT#1, vari.controlCylNum, UINT#4);
    FOR index := 0 TO 3 DO
      sensorOff[index] := FALSE;
      IF index < vari.controlCylNum THEN
        sensorOn[index] := TRUE;
      ELSE
        sensorOn[index] := FALSE;
      END_IF;
    END_FOR;
    	
    //画面显示
	vari.display := vari.stationNo >0;

    //气缸显示模式=气缸控制的数量
    vari.displayCylNum := vari.controlCylNum;
    
    
	
  
//-----------------------------------------------------------------------------------//
END_ACTION

END_FUNCTION_BLOCK

// ---- Standard/Unit/06 Axis/FB_Axis_RD.TcPOU
FUNCTION_BLOCK FB_Axis_RD
VAR_INPUT
END_VAR
VAR_OUTPUT
END_VAR

VAR_IN_OUT
machine : UDT_Machine_RD; //
station : UDT_Station_RD; //
vari : UDT_AxisVar_RD; //
data : UDT_AxisData_RD; //
  
END_VAR

VAR
safetyPermit : BOOL; //
operatePermit : BOOL; //
mcPower : MC_Power; //
mcReadStatus : MC_ReadStatus;//
mcMoveJog : MC_Jog; //
mcHome : MC_Home; //
mcMoveAbs : MC_MoveAbsolute; //
mcMoveAbs2 : MC_MoveAbsolute; //
mcMoveRel : MC_MoveRelative; //
mcMoveModulo :MC_MoveModulo;//
mcReset : MC_Reset; //
mcStop : MC_Stop; //
mcHalt : MC_Halt;//
mcVelocity					: MC_MoveVelocity;		//
inPositionTimer : TON; //
brakeOpenTimer : TON; //
brakeCloseTimer : TON; //
homehmiTimer : TON; //
autoTipsTimer : TON; //
notPowerOnTimer : TON; //
notHomeTimer : TON; //
velocityTimer	: TON;					//
posTeachTimer :TON;
isBrakeOpenTimer : BOOL; //
isBrakeCloseTimer : BOOL; //
isAutoTipsTimer : BOOL; //
powerhmiCache : BOOL; //
brakehmiCache : BOOL; //
movehmiCache : BOOL; //
jogForward : BOOL; //
jogBackward : BOOL; //
moveNo : UINT; //
moveNoCache : UINT; //
moveVelo : REAL; //
index : UINT; //
moduloPresetPos : UINT; //模长控制预置定位数量
notMovePermitManualTipCache : UINT; //
moduloCalculate : FB_ModuloCalculate_RD; //

mcReadAxisParameter : MC_ReadParameterSet; //读取NC参数设置功能块
mcWriteParameterPersistent	: MC_WriteParameterPersistent;	//修改NC参数功能块
parameter				: ST_AxisParameterSet;	//NC参数设置
fbSoEReset			: FB_SoEReset;			//动器复位功能块

mcMoveAdditive : MC_MoveAdditive;


activated : Bool; //
calibratePos : REAL; //
error : BOOL; //
homed : BOOL; //
ncErrCode : UDINT; //
driverErrID : UDINT; //
jogft:F_TRIG;
 
  
END_VAR

VAR CONSTANT
END_VAR

VAR PERSISTENT
  homeOffset :REAL;
END_VAR

SetUp();
Servo();
Alarm();
General();
Modulo();
Manual();
Power();
Brake();
Reset();
Home();
StopAndHalt();
JOG();
Movement();
InPosition();
Velocity();
ManualTip();
AutoTip();
AutoReturn();
Status();
Display();
Additive();

ACTION Additive:
mcMoveAdditive(
	Axis:= vari.axis, 
	Execute:= vari.additiveAuto, 
	Distance:= vari.additiveDistance, 
	Velocity:= vari.additiveVelo, 
	Acceleration:= data.acceleration, 
	Deceleration:= data.deceleration, 
	Jerk:= , 
	BufferMode:= , 
	Options:= , 
	Done=> , 
	Busy=> , 
	Active=> , 
	CommandAborted=> , 
	Error=> , 
	ErrorID=> );
END_ACTION

ACTION Alarm:
//---------------------------------------Alarm-------------------------------------------------------//
    
    //报警复位
    IF vari.resethmi OR machine.reset THEN
      vari.error := FALSE;
      vari.driverErrID := 0;
      vari.ncErrID := 0;
    END_IF;

    //伺服错误中
    IF error OR ncErrCode <> 0 OR driverErrID <> 0 THEN
		vari.error := TRUE;
		vari.ncErrID := ncErrCode;
    vari.driverErrID := driverErrID;
    END_IF;
    vari.alarming := vari.error OR vari.warning;
    //反馈报警中
    IF vari.alarming THEN
      machine.alarmCount := machine.alarmCount+1; 
      station.report.alarming := TRUE;
    END_IF;
   
  //----------------------------------------------------------------------------------------------------//
END_ACTION

ACTION AutoReturn:
 //---------------------------------------AutoReturn------------------------------------------------//
    //自动回位
    IF vari.autoReturnEnable THEN
      IF vari.notInPosAutoTip > 0
        AND vari.notInPosAutoTip = vari.moveAutoNoCache
        AND machine.autoMode
        AND NOT station.running
        AND vari.ready
        AND NOT vari.busy
        AND (ABS(vari.actPos - data.movePos[vari.moveAutoNoCache]) <= vari.autoReturnScope //位置偏差在自动回位范围之内
        OR vari.movePermits[vari.moveAutoNoCache] AND vari.autoReturnPermit) //或者定位条件满足
      THEN
        vari.autoReturnAllow := TRUE;
        IF machine.reset THEN
          moveNo := vari.moveAutoNoCache;
          vari.autoReturning := TRUE;
        ELSE
          vari.autoReturning := FALSE;
        END_IF;
      ELSIF NOT vari.busy THEN
        vari.autoReturnAllow := FALSE;
        vari.autoReturning := FALSE;
      END_IF;
    ELSE
      vari.autoReturnAllow := FALSE;
      vari.autoReturning := FALSE;
    END_IF;
  //----------------------------------------------------------------------------------------------------//
END_ACTION

ACTION AutoTip:
//---------------------------------------AutoTip----------------------------------------------------//
    
    // 伺服未使能提示
    notPowerOnTimer(IN := vari.powerAuto AND NOT vari.isPowerOn,
                  PT := T#0.3S,
                  Q  => vari.notPowerOnAutoTip); //伺服未使能延时
 
    // 伺服未回原点提示
    notHomeTimer(IN := NOT vari.homeDone,
                  PT := T#0.3S,
                  Q  => vari.notHomeAutoTip); //伺服未回原点延时
    
    //伺服不在位自动提示延时,伺服未动作且工站未运行时
    autoTipsTimer(IN := NOT vari.busy AND NOT station.running,
                   PT := T#0.5S,
				   Q=>isAutoTipsTimer);
    IF isAutoTipsTimer
      AND NOT vari.inPos[vari.moveAutoNoCache]
      AND NOT vari.absOrRel[vari.moveAutoNoCache]
      AND vari.moveAutoNoCache > 0
      AND vari.moveAutoNoCache <= vari.movePosNum
    THEN
      vari.notInPosAutoTip := vari.moveAutoNoCache;
    ELSE
      vari.notInPosAutoTip := 0;
    END_IF;
    
    // 自动提示
    vari.autoTip := vari.notHomeAutoTip OR vari.notPowerOnAutoTip OR vari.notInPosAutoTip > 0;

    // 反馈工站自动提示
    IF vari.autoTip THEN
      station.report.autoTip := TRUE;
    END_IF;
    
  //----------------------------------------------------------------------------------------------------//
END_ACTION

ACTION Brake:
//---------------------------------------Brake -------------------------------------------------------//
    
    vari.brake := vari.brakeManual OR vari.isPowerOn;//刹车正常打开输出
    vari.brakeForced := vari.brakeManual;//刹车强制打开输出
    brakeCloseTimer(IN := NOT vari.brakeForced,
                     PT := T#0.3S,
					 Q=>isBrakeCloseTimer);
    brakeOpenTimer(IN := vari.brake,
                    PT := T#0.3S,
					Q=>isBrakeOpenTimer);
    
  //----------------------------------------------------------------------------------------------------//
END_ACTION

ACTION Display:
 
    //---------------------------------------Display------------------------------------------------------//
      
      //禁止图标显示
      vari.powerForbidIcon := NOT machine.manualMode OR NOT vari.powerAllow;
      vari.homeForbidIcon := NOT machine.manualMode OR NOT vari.homeAllow;
      vari.moveForbidIcon := NOT machine.manualMode OR NOT vari.moveAllow OR NOT vari.movePermits[vari.movehmiNo];
      vari.jogForwardForbidIcon := NOT machine.manualMode OR NOT vari.jogForwardAllow;
      vari.jogBackwardsForbidIcon := NOT machine.manualMode OR NOT vari.jogBackwardsAllow;
      vari.brakeForbidIcon := NOT vari.brakeAllow AND vari.brakeEnable;
      
      //刹车按钮指示状态
      IF NOT vari.brakeEnable THEN
        vari.brakeState := 2;
      ELSIF vari.brake THEN
        vari.brakeState := 1;
      ELSE
        vari.brakeState := 0;
      END_IF;
      
    //----------------------------------------------------------------------------------------------------//
END_ACTION

ACTION General:
//---------------------------------------General-----------------------------------------------------//

    //已回原点
    vari.homeDone := homed OR TRUE;
    
    //安全条件
    safetyPermit := machine.eStop
    AND machine.safety
    AND machine.airOn
    AND machine.allDoorClosed;
    
    //伺服可操作
    operatePermit := safetyPermit
    AND NOT vari.alarming;
    
    //伺服忙信号
    vari.busy :=
    mcReset.Busy
    OR mcMoveJog.Busy
    OR mcMoveAbs.Busy
    OR mcMoveRel.Busy	
    OR mcHome.Busy
    OR mcMoveModulo.Busy
    OR mcVelocity.Busy;
	
    //伺服准备好信号
    vari.ready := operatePermit
    AND vari.isPowerOn
    AND isBrakeOpenTimer;
    
    //伺服On允许操作
    vari.powerAllow := operatePermit AND NOT vari.brakeManual;
    //回原点允许操作
    vari.homeAllow :=  vari.homePermit;
    //定位允许操作
    vari.moveAllow := vari.ready AND vari.movePermit;
    //JOG+允许操作
    vari.jogForwardAllow := vari.ready AND vari.jogForwardPermit AND NOT vari.lsp;
    //JOG-允许操作
    vari.jogBackwardsAllow := vari.ready AND vari.jogBackwardsPermit AND NOT vari.lsn;
    //刹车允许操作
    vari.brakeAllow := machine.manualMode AND NOT vari.isPowerOn AND vari.brakeEnable;
    //回原点按钮显示
    vari.homeDisplay := NOT vari.homeDone OR data.homeDisplay;
    
    
  //----------------------------------------------------------------------------------------------------//
END_ACTION

ACTION Home:
  //---------------------------------------Home-------------------------------------------------------//
    //回原点执行   
  
IF vari.homeMode = 0 THEN
  IF (vari.homeManual OR vari.homeInit) AND vari.homePermit THEN 
    homeOffset := LREAL_TO_REAL(REAL_TO_LREAL(0.0-vari.actPos)+parameter.fEncOffset);
    mcWriteParameterPersistent.Execute:=TRUE;
	END_IF
  IF ABS(REAL_TO_LREAL(homeOffset)-parameter.fEncOffset)>0.01 THEN
    IF NOT mcWriteParameterPersistent.Busy 
		  AND NOT mcWriteParameterPersistent.Error
		  AND NOT mcWriteParameterPersistent.Execute
	  THEN
		  mcWriteParameterPersistent.Execute:=TRUE;
	  END_IF	
  END_IF

  mcWriteParameterPersistent(
    Axis:= vari.axis, 
    Execute:= , 
    ParameterNumber:= MC_AxisParameter.AxisEncoderOffset, 
    Value:= homeOffset, 
    Done=> , 
    Busy=> , 
    Error=> , 
    ErrorID=> );

  mcWriteParameterPersistent.Execute:=FALSE;
 
ELSIF vari.homeMode = 1 THEN
  
  mcHome(
        	Axis:=vari.axis,
	        Execute:=(vari.homeManual OR vari.homeInit) AND vari.homePermit,
          bCalibrationCam:= , 
	        Busy=>vari.homing,
        );
  vari.homeInit := FALSE;

END_IF
  


    
    
      //----------------------------------------------------------------------------------------------------//
END_ACTION

ACTION InPosition:
  //---------------------------------------In Position--------------------------------------------------//
    
    //伺服到位延时
    inPositionTimer(IN := vari.ready AND NOT vari.busy,
                     PT := vari.inPosTime);
    //根据设定的伺服到位精度显示伺服位置
    FOR index := 1 TO vari.movePosNum DO
      IF NOT vari.modulo.enable
        OR index > moduloPresetPos
      THEN
        vari.inPos[index] := inPositionTimer.Q AND ABS(vari.actPos - data.movePos[index]) <= vari.inPosScope;
      END_IF;
    END_FOR;
    
    vari.inPosNo := FUN_AryBitOnNum_RD(vari.inPos);
  //----------------------------------------------------------------------------------------------------//
END_ACTION

ACTION JOG:
//---------------------------------------JOG  --------------------------------------------------------//
    //点动+执行
    jogForward := vari.jogForwardAllow
    AND NOT jogBackward
    AND (vari.jogForwardhmi
    AND machine.manualMode
    OR vari.jogForwardAuto);
    
    //点动-执行
    jogBackward := vari.jogBackwardsAllow
    AND NOT jogForward
    AND (vari.jogBackwardshmi
    AND machine.manualMode
    OR vari.jogBackwardsAuto);
	
 IF  data.jogDistance = 0 THEN
   mcMoveJog.Mode := MC_JOGMODE_CONTINOUS;
 ELSE
   mcMoveJog.Mode := MC_JOGMODE_INCHING;
 END_IF
  
	mcMoveJog(
	Axis:=vari.axis,
	JogForward:=jogForward,
	JogBackwards:=jogBackward,
	Mode:=,
	Position:= data.jogDistance,
	Velocity:=REAL_TO_LREAL(data.jogVelo),
	Acceleration:=data.acceleration,
	Deceleration:=data.deceleration,
	Jerk:=,
	Done=>,
	Busy=>,
	Active=>,
	CommandAborted=>,
	Error=>,
	ErrorID=>
);
  
jogft(CLK:= vari.jogForwardhmi OR vari.jogBackwardshmi, Q=> );              
IF  mcMoveJog.Mode = MC_JOGMODE_INCHING AND NOT vari.Axis.Status.NotMoving THEN
  IF jogft.Q =TRUE THEN  
    vari.haltAuto :=TRUE;
   END_IF 
END_IF
IF mcHalt.Done THEN 
  vari.haltAuto :=FALSE;
END_IF
 
       
                
	  vari.jogForwardAuto := FALSE;
    vari.jogBackwardsAuto := FALSE;
	
  //----------------------------------------------------------------------------------------------------//
END_ACTION

ACTION Manual:
//---------------------------------------Manual-----------------------------------------------------//
    
    IF machine.manualMode THEN//只有在手动模式且hmi操作/显示激活
      
      //伺服On
      IF powerhmiCache AND NOT vari.powerhmi AND vari.powerAllow THEN
        vari.powerManual := NOT vari.powerManual;
      END_IF;
      powerhmiCache:=vari.powerhmi;
      //手动刹车
      IF brakehmiCache AND NOT vari.brakehmi AND vari.brakeAllow THEN
        vari.brakeManual := NOT vari.brakeManual;
      END_IF;
      brakehmiCache:= vari.brakehmi;
      //手动回原点	  
      homehmiTimer(IN := vari.homehmi AND vari.homeAllow,
                    PT := T#1S,
					Q=>vari.homeManual);
      
      //手动定位

      IF movehmiCache AND NOT vari.movehmi
        AND vari.moveAllow
        AND vari.moveAutoNo = 0
      THEN
        moveNo := vari.movehmiNo;
      END_IF;
      movehmiCache := vari.movehmi;
    END_IF;
    
    
    posTeachTimer(IN:= vari.posTeach, PT:=T#1S , Q=> , ET=> );   
    IF NOT vari.modulo.enable THEN
      IF posTeachTimer.Q THEN
        data.movePos[vari.movehmiNo]:=vari.actPos;
		  END_IF
		END_IF


    
    vari.targetDistance := data.movePos[vari.movehmiNo];
    vari.targetVelocity := data.manualVelo ;
  //----------------------------------------------------------------------------------------------------//
END_ACTION

ACTION ManualTip:
//---------------------------------------ManualTip -------------------------------------------------//
    
    // 整机手动提示           
    IF vari.powerhmi
      OR vari.movehmi
      OR vari.homehmi
      OR vari.jogForwardhmi
      OR vari.jogBackwardshmi
      OR vari.brakehmi AND vari.brakeEnable AND NOT vari.brakeAllow
    THEN
      machine.presetManualTips[0] := NOT machine.eStop;     //急停中,无法操作
      machine.presetManualTips[1] := NOT machine.safety;    //安全条件不满足,无法操作
      machine.presetManualTips[2] := NOT machine.allDoorClosed;  //安全门未锁好,无法操作
      machine.presetManualTips[3] := NOT machine.airOn;     //气压不足,无法操作
      machine.presetManualTips[4] := NOT machine.manualMode;//不在手动模式,无法操作
    END_IF;
    
    //手动提示复位
    IF machine.tipReset
      OR (notMovePermitManualTipCache <> 0
      AND vari.notMovePermitManualTip = 0)
    THEN
      vari.notMovePermitManualTip := 0;
	  vari.notPowerOnManualTip:=FALSE;
	  vari.unableBrakeManualTip:=FALSE;
	   vari.unablePowerOnManualTip:=FALSE; 
    END_IF;
    notMovePermitManualTipCache := vari.notMovePermitManualTip;
    
    //手动提示
    IF NOT vari.isPowerOn
      AND (vari.movehmi
      OR vari.jogForwardhmi
      OR vari.jogBackwardshmi)
    THEN
	 vari.notPowerOnManualTip:=TRUE;//  伺服未使能无法操作
    ELSIF vari.brakehmi AND vari.brakeEnable AND vari.isPowerOn THEN
      vari.unableBrakeManualTip:=TRUE; //  伺服ON时无法操作刹车
    ELSIF vari.powerhmi AND operatePermit AND vari.brakeManual THEN
      vari.unablePowerOnManualTip:=TRUE;  // 刹车手动打开时无法操作伺服ON   
    ELSIF vari.movehmi AND (NOT vari.movePermit OR NOT vari.movePermits[vari.movehmiNo]) THEN
      vari.notMovePermitManualTip := vari.movehmiNo;  // 定位条件不足手动提示
    END_IF;
    
    // 手动提示
    vari.manualTip := vari.notMovePermitManualTip <> 0
	OR vari.notPowerOnManualTip
	OR vari.unableBrakeManualTip
	OR vari.unablePowerOnManualTip;
	
    // 反馈工站手动提示
    IF vari.manualTip THEN
      station.report.manualTip := TRUE;
    END_IF;
    
  //----------------------------------------------------------------------------------------------------//
END_ACTION

ACTION Modulo:
//--------------------------------- ModuloCalculate------------------------------------------------//
  
	IF vari.modulo.enable THEN
		IF vari.modulo.mode =0 THEN
			moduloCalculate(actPos       		:= vari.actPos,
					                    modulo       		:= vari.modulo,
					                    calibratePos 	:= data.movePos[1]);
			vari.movePosNum := MAX(vari.movePosNum, moduloPresetPos);
			vari.absOrRel[1] := FALSE;
			vari.absOrRel[2] := FALSE;
			vari.absOrRel[3] := FALSE;
			vari.absOrRel[4] := FALSE;
			vari.absOrRel[5] := FALSE;
			vari.absOrRel[6] := FALSE;
			IF vari.moveAutoNoCache = 2
				OR vari.moveAutoNoCache = 3
				OR vari.moveAutoNoCache = 5
				OR vari.moveAutoNoCache = 6
			THEN
				vari.moveAutoNoCache := 4;
			END_IF;
			data.movePos[2] := vari.modulo.closestPos;   //最近分割点位置
			data.movePos[3] := vari.modulo.autoNextPos;  //下一自动分割点位置
			data.movePos[4] := vari.modulo.autoPos;      //自动分割点位置
			data.movePos[5] := vari.modulo.nextPos;      //下一分割点位置
			data.movePos[6] := vari.modulo.previousPos;  //上一分割点位置

			vari.inPos[1] := vari.modulo.inCalibratePos;     //在标定分割点位置
			vari.inPos[2] := vari.modulo.inClosestPos;  //在分割点位置
			vari.inPos[3] := vari.modulo.inAutoNextPos; //在下一自动分割点位置
			vari.inPos[4] := vari.modulo.inAutoPos;     //在自动分割点位置
			vari.inPos[5] := FALSE;
			vari.inPos[6] := FALSE;

		ELSIF  vari.modulo.mode =1 THEN
			moduloCalculate(actPos       		:= vari.actPos,
					            modulo       		:= vari.modulo,
					            calibratePos 	:= calibratePos);
			vari.movePosNum := MAX(vari.movePosNum, moduloPresetPos);
			vari.absOrRel[1] := FALSE;
			vari.absOrRel[2] := FALSE;
			vari.absOrRel[3] := FALSE;
			vari.absOrRel[4] := TRUE;
			
			IF vari.moveAutoNoCache = 2
				OR vari.moveAutoNoCache = 3
				OR vari.moveAutoNoCache = 4
			THEN
				vari.moveAutoNoCache := 1;
			END_IF;
			data.movePos[1] := vari.modulo.closestPos;   //最近分割点位置
			data.movePos[2] := vari.modulo.nextPos;      //下一分割点位置
			data.movePos[3] := vari.modulo.previousPos;  //上一分割点位置
			vari.inPos[1] := vari.modulo.inClosestPos;  //在分割点位置
			vari.inPos[2] := FALSE;
			vari.inPos[3] := FALSE;
			vari.inPos[4] := FALSE;
			
		ELSIF  vari.modulo.mode =2 THEN
			moduloCalculate(actPos       		:= vari.actPos,
					            modulo       		:= vari.modulo,
					            calibratePos 	:= calibratePos);
			vari.movePosNum := MAX(vari.movePosNum, moduloPresetPos);
			vari.absOrRel[1] := FALSE;
			data.movePos[1] := vari.modulo.closestPos;   //最近分割点位置
			vari.inPos[1] := vari.modulo.inClosestPos;  //在分割点位置
			
		END_IF;
	END_IF;
  
  
  (**)
 
  //----------------------------------------------------------------------------------------------------//
END_ACTION

ACTION Movement:
//---------------------------------------Move-------------------------------------------------------//
    //自动定位
    IF vari.moveAutoNo > 0 THEN
      moveNo := vari.moveAutoNo;
    END_IF;
    // 定位执行
    IF vari.moveAllow
      AND moveNo > 0
      AND moveNoCache <> moveNo
      AND (vari.movePermits[moveNo] OR vari.autoReturning)
    THEN
      IF NOT machine.autoMode THEN
        moveVelo := data.manualVelo;  //手动速度
      ELSE
        IF vari.differentVelo = 0.0 THEN//当设定单独定位速度时以单独定位速度执行，否则按自动速度执行
          moveVelo := data.autoVelo;  //自动速度
        ELSE
          moveVelo := vari.differentVelo; //单独定位速度
        END_IF;
      END_IF;
      
      
          IF NOT vari.modulo.enable THEN    
              IF NOT vari.absOrRel[moveNo] THEN
                // 绝对定位时
                  mcMoveAbs(axis := vari.axis,
                            Execute := TRUE,
                            Position := data.movePos[moveNo],
                            Velocity := moveVelo,
                            Acceleration := data.acceleration,
                            Deceleration := data.deceleration
                            );
              IF vari.moveAutoNo > 0 THEN //自动定位编号暂存写入相应值
                vari.moveAutoNoCache := vari.moveAutoNo;
              END_IF;
            ELSE
                // 相对定位时
                  mcMoveRel(axis := vari.axis,
                            Execute := TRUE,
                            Distance := data.movePos[moveNo],
                            Velocity := moveVelo,
                            Acceleration := data.acceleration,
                            Deceleration := data.deceleration
                        );
                vari.moveAutoNoCache := 0; //自动定位编号暂存写入0
             END_IF;
          ELSIF vari.modulo.enable THEN
                  mcMoveModulo(
                          Axis:= vari.axis, 
                          Execute:= TRUE, 
                          Position:= data.movePos[moveNo], 
                          Velocity:= moveVelo, 
                          Acceleration:= data.acceleration, 
                          Deceleration:= data.deceleration, 
                          Direction:= MC_Shortest_Way, 
                        );    
              IF vari.moveAutoNo > 0 THEN //自动定位编号暂存写入相应值
                vari.moveAutoNoCache := vari.moveAutoNo;
              END_IF;    
        END_IF;
 END_IF;   
    
    moveNoCache := moveNo;
    moveNo := 0;
    vari.moveAutoNo := 0;
    vari.differentVelo := 0.0;
		mcMoveAbs   (axis    := vari.axis,
	               			Execute := FALSE);
	  mcMoveRel   (axis    := vari.axis,
	               			Execute := FALSE);
    mcMoveModulo(axis := vari.axis,
	                    Execute := FALSE);                     
                      

  //----------------------------------------------------------------------------------------------------//*)
END_ACTION

ACTION Power:
  //---------------------------------------Power------------------------------------------------------//
    
    IF vari.powerInit THEN
      vari.powerAuto := TRUE;
      vari.powerManual := FALSE;
      vari.powerInit := FALSE;
    END_IF;
	
	mcPower(
	Axis:=vari.axis,
	Enable:=operatePermit
					AND isBrakeCloseTimer
					 AND (vari.powerAuto XOR vari.powerManual),
	Enable_Positive:=operatePermit,
	Enable_Negative:=operatePermit,
	Override:=vari.Override,
	BufferMode:=,
	Options:=,
	Status=>vari.isPowerOn,
	Busy=>,
	Active=>,
	Error=>,
	ErrorID=>
);

  //----------------------------------------------------------------------------------------------------//
END_ACTION

ACTION Reset:
  //---------------------------------------Reset-------------------------------------------------------//
    //异常复位
   mcReset.Execute := (vari.resethmi OR machine.reset) AND (vari.error OR vari.warning);    	
	 mcReset(axis := vari.axis);

  //----------------------------------------------------------------------------------------------------//
  
  
  //	NC轴错误复位
fbSoEReset(
	NetId:=,
	Execute:= (vari.resethmi OR machine.reset) AND (vari.error OR vari.warning),
	Timeout:=,
	Axis:=vari.axis,
	Busy=>,
	Error=>,
	AdsErrId=>,
	SercosErrId=>
);

//	驱动器错误复位
mcReset(
	Axis:=vari.axis,
	Execute:= (vari.resethmi OR machine.reset) AND (vari.error OR vari.warning),
	Done=>,
	Busy=>,
	Error=>,
	ErrorID=>
);
END_ACTION

ACTION Servo:
 //---------------------------------------Servo-----------------------------------------------------//
   IF  NOT vari.modulo.enable THEN
     vari.actPos := LREAL_TO_REAL(vari.axis.NcToPlc.ActPos);
     ELSE
     vari.actPos := LREAL_TO_REAL(vari.axis.NcToPlc.ModuloActPos);  
	 END_IF;

     
    
    vari.actVelo := LREAL_TO_REAL(vari.axis.NcToPlc.ActVelo);
    vari.actTorque := LREAL_TO_REAL(vari.axis.NcToPlc.ActTorque);
        
    //正负极限位置
	//vari.lsn := vari.axis.DrvStatus.N_OT;
	//vari.lsp := vari.axis.DrvStatus.P_OT;
	//vari.dog := vari.axis.Status.Homed;
	error:= vari.axis.Status.Error OR vari.axis.Status.DriveDeviceError;
	ncErrCode:=vari.axis.NcToPlc.ErrorCode;
  driverErrID:=vari.axis.Status.ErrorID;
	homed:=vari.axis.Status.Homed;
  
  
	mcReadAxisParameter(
	Parameter:=parameter,
	Axis:=vari.axis,
	Execute:=activated,
	Done=> , 
	Busy=> , 
	Error=> , 
	ErrorID=>);
  
  mcReadStatus(
	Axis:= vari.axis, 
	Enable:= activated, 
 );

  
	
  //----------------------------------------------------------------------------------------------------//
END_ACTION

ACTION SetUp:
//---------------------------------------SetUp------------------------------------------------------//
    
	//第一个扫描周期
	IF NOT activated THEN
		activated 		:=TRUE;
		vari.autoReturnEnable		:=TRUE;
		vari.jogForwardPermit		:=TRUE;
		vari.jogBackwardsPermit	:=TRUE;
		vari.homePermit			:=TRUE;
		vari.movePermit			:=TRUE;
    vari.VelocityPermit :=TRUE;
		vari.inPosScope			:=0.03;
		vari.autoReturnScope	:=2.0;

		IF vari.modulo.mode =0 THEN
			moduloPresetPos:=6;		
		ELSIF  vari.modulo.mode =1 THEN
			moduloPresetPos:=4;
		ELSIF  vari.modulo.mode =2 THEN
			moduloPresetPos:=1;
		END_IF;
		
		FOR index :=0 TO SIZEOF(vari.inPos) -1 DO
			vari.movePermits[index]:=TRUE;
		END_FOR;		
		
		//伺服单位赋初值
		vari.posUnit			:='mm';
		vari.veloUnit			:='mm/s';
		vari.accDecUnit	  :="mm/s²";
		//伺服速度赋初值
    moveVelo := 1;
		IF data.manualVelo <= 0.0 THEN
		  data.manualVelo := 5.0;
		END_IF;
		IF data.autoVelo <= 0.0 THEN
		  data.autoVelo := 10.0;
		END_IF;
		IF data.jogVelo <= 0.0 THEN
		  data.jogVelo := 1.0;
		END_IF;
		//伺服加减速度赋初值
		IF data.acceleration = 0.0 THEN
		  	data.acceleration := 30000.0;
		END_IF;
		IF data.deceleration = 0.0 THEN
		  	data.deceleration := 30000.0;
		END_IF;
	END_IF;
 
	// 显示在hmi上面
	vari.display := vari.stationNo >0;
       
    //检查定位位置数量
   vari.movePosNum :=	MIN(vari.movePosNum,
												(SIZEOF(vari.inPos)-1));
END_ACTION

ACTION Status:
    
    //---------------------------------------Status----------------------------------------------------//
      // 伺服状态显示
      IF vari.error THEN
        vari.status := 0;//伺服报警中
      ELSIF vari.warning THEN
        vari.status := 1;//伺服警告中
      ELSIF NOT vari.isPowerOn THEN
        vari.status := 2;//伺服OFF
      ELSIF vari.isPowerOn THEN
        vari.status := 3;//伺服准备好
      END_IF;
      IF NOT vari.homeDone THEN
        vari.status := 4;//伺服未回原点
      END_IF;
      IF mcHome.Busy THEN
        vari.status := 5;//伺服回原点中
      END_IF;
      IF vari.lsp THEN
        vari.status := 6;//伺服正极限
      ELSIF vari.lsn THEN
        vari.status := 7;//伺服负极限
      END_IF;
    //----------------------------------------------------------------------------------------------------//
END_ACTION

ACTION StopAndHalt:
  //---------------------------------------Stop--------------------------------------------------------//
    //停止伺服
    vari.stopManual := vari.stophmi AND operatePermit;
    
	  mcStop(	axis := vari.axis,
			   	  Execute := NOT vari.isPowerOn OR NOT safetyPermit OR vari.stopAuto OR vari.stopManual,
            Deceleration:=data.deceleration , 
	          Jerk:=, );
            
  //---------------------------------------Halt--------------------------------------------------------//
     
    //暂停伺服
  vari.haltManual := vari.halthmi AND operatePermit;

	  mcHalt(	axis := vari.axis,
			   	  Execute := NOT vari.isPowerOn OR NOT safetyPermit OR vari.haltAuto OR vari.haltManual,
	          Deceleration:= data.deceleration, 
	          Jerk:=, );
END_ACTION

ACTION Velocity:
  vari.VelocityAllow := vari.ready AND vari.VelocityPermit ;

//	速度定位超时
velocityTimer(
	IN:=vari.velocityBusy,
	PT:=T#20S,
	Q=>, ET=>
);

    
    
IF velocityTimer.Q
	OR NOT vari.ready
  OR vari.InVelocity
THEN
	vari.velocityAuto:=FALSE;
	vari.velocityHmi:=FALSE;
END_IF


mcVelocity(
	Axis:=vari.axis,
	Execute:=vari.VelocityAllow AND (vari.velocityHmi AND machine.manualMode OR vari.velocityAuto),
	Velocity:=vari.Velocity,
	Acceleration:=data.acceleration,
	Deceleration:=data.deceleration,
	Jerk:=,
	Direction:=,
	BufferMode:=,
	Options:=,
	InVelocity=>vari.InVelocity,
	Busy=>vari.velocityBusy,
	Active=>,
	CommandAborted=>,
	Error=>vari.velocityError,
	ErrorID=>vari.velocityErrorID
);
END_ACTION

END_FUNCTION_BLOCK

// ---- Standard/Unit/06 Axis/FB_ModuloCalculate_RD.TcPOU
FUNCTION_BLOCK FB_ModuloCalculate_RD
VAR_INPUT
actPos : REAL; // 当前坐标
END_VAR
VAR_OUTPUT
END_VAR
VAR_IN_OUT

modulo : UDT_ModuloProperty_RD; //
calibratePos : Real; // 设置标定位置坐标

END_VAR
VAR
calibratePosCache : REAL; //标定位置缓存
calibrateOffsetCache : Real; //标定位置偏移缓存
offset : Real; //偏移坐标
actPosModAbs : Real; // 当前模长位置
actDis : Real; //
closestDis : Real; //

END_VAR

ACT();

ACTION ACT:
IF modulo.factor > 0
  AND modulo.divisor >=1
  AND modulo.stepPoint > 0
THEN
  IF calibratePosCache <> calibratePos
    OR calibrateOffsetCache <> modulo.calibrateOffset
    OR calibratePosCache = 0.0
  THEN
    calibratePos :=
    Modabs
    (calibratePos,
     modulo.factor
    );
    
    offset := modulo.calibrateOffset +
    LREAL_TO_REAL(Modabs(calibratePos,modulo.factor / modulo.divisor));
    
    calibratePosCache := calibratePos;
    calibrateOffsetCache := modulo.calibrateOffset;
  END_IF;
  
  actPosModAbs :=
  LREAL_TO_REAL(Modabs(actPos - offset,modulo.factor));
  
  modulo.actPoint:= LINT_TO_INT(TRUNC(actPosModAbs * modulo.divisor / modulo.factor));
  
  actDis := actPosModAbs - modulo.actPoint * modulo.factor / modulo.divisor;
  
  IF actDis < modulo.factor / modulo.divisor / 2 THEN
    modulo.closestPoint := modulo.actPoint;
    closestDis := actDis;
  ELSE
    modulo.closestPoint := REAL_TO_INT
    (LREAL_TO_REAL(Modabs(modulo.actPoint + 1,modulo.divisor))
    );
    closestDis := MIN
    (
     LREAL_TO_REAL(Modabs(actPosModAbs- modulo.closestPoint * modulo.factor / modulo.divisor,modulo.factor)),
     
     LREAL_TO_REAL(Modabs(modulo.closestPoint * modulo.factor / modulo.divisor - actPosModAbs,modulo.factor)));
  END_IF;
  
  modulo.inClosestPos := ABS(closestDis)
  <= ABS(modulo.tolerance);
  
  modulo.previousPoint := REAL_TO_INT
  (LREAL_TO_REAL(Modabs(SEL(modulo.inClosestPos,modulo.actPoint,DINT_TO_INT(modulo.closestPoint - modulo.stepPoint)),modulo.divisor)));

  modulo.nextPoint := REAL_TO_INT
  (LREAL_TO_REAL(Modabs(SEL(modulo.inClosestPos,modulo.actPoint,modulo.closestPoint) + modulo.stepPoint,modulo.divisor)));
  
  modulo.autoPoint := REAL_TO_INT
  (LREAL_TO_REAL(Modabs(modulo.autoPoint, modulo.divisor)));
  
  modulo.autoNextPoint := REAL_TO_INT
  (LREAL_TO_REAL(Modabs(modulo.autoPoint + modulo.stepPoint,modulo.divisor)));
  
  modulo.closestPos := offset
  + modulo.closestPoint * modulo.factor / modulo.divisor;
  
  modulo.previousPos := 
  LREAL_TO_REAL(Modabs(offset+ modulo.previousPoint * modulo.factor / modulo.divisor,modulo.factor));
  
  modulo.nextPos := offset
  + modulo.nextPoint * modulo.factor / modulo.divisor;
  
  modulo.autoPos := offset
  + modulo.autoPoint * modulo.factor / modulo.divisor;
  
  modulo.autoNextPos := offset
  + modulo.autoNextPoint * modulo.factor / modulo.divisor;
  
  modulo.inCalibratePos := ABS(actPos - calibratePos) <= modulo.tolerance
  OR ABS(actPos - calibratePos) >= modulo.factor - modulo.tolerance;
  
  modulo.inAutoPos := modulo.inClosestPos
  AND modulo.closestPoint = modulo.autoPoint;
  modulo.inAutoNextPos := modulo.inClosestPos
  AND modulo.closestPoint = modulo.autoNextPoint;
ELSE
  modulo.inClosestPos := 0;
  modulo.inCalibratePos := 0;
  modulo.inAutoPos := 0;
  modulo.inAutoNextPos := 0;
END_IF;
END_ACTION

END_FUNCTION_BLOCK

// ---- Standard/FUN/FUN_AryBitOnNum_RD.TcPOU
FUNCTION FUN_AryBitOnNum_RD : UINT
VAR_IN_OUT
 IN : ARRAY[*] OF BOOL;
END_VAR
VAR
    index : uINT;
END_VAR

FUN_AryBitOnNum_RD:=0;
FOR index:=0 TO SIZEOF(IN)-1 DO
	IF IN[index] THEN
    FUN_AryBitOnNum_RD := index ;
	END_IF;	
END_FOR;

END_FUNCTION

// ---- Standard/Public/06 Produce/FB_Produce.TcPOU
FUNCTION_BLOCK FB_Produce
VAR_IN_OUT
machine : UDT_Machine_RD; //
stations : ARRAY[*] OF UDT_Station_RD; //
vari : UDT_ProduceVar_RD; //
data : UDT_ProduceData_RD; //
badVar : ARRAY[*] OF UDT_BadVar_RD; //
badData : ARRAY[*] OF UDT_BadData_RD; //
lastProduce : UDT_ProduceDataRecord_RD; //
END_VAR

VAR
goodExecuteCache : ARRAY[0..99] OF BOOL; // 不良触发缓存
activated : Bool; //
badExecuteCache : Array[0..99] of Bool; // 缓存不良数量
badList : Array[0..99] of Int; // 不良排序列表
maxValue : DInt; //
minValue : DInt; //
badTypeNum : Int; // 报警推送
pushAlarmNo : UInt; // 清零定时器
clearTimer : TON; // 设定定时器
resetCache : Bool; //
index : DInt; //
index1 : DInt; //
temp : DInt; //
totalBad : DInt; //
badMax : DInt; //
No : INT; //
test  : ARRAY[0..5] OF DINT;
lastIndex : DINT := 1;
index3 : INT;
numListPOINT : POINTER TO DINT;
END_VAR

VAR CONSTANT
MAX_CONTINUOUS : INT :=99; // 最大连续不良报警数量
MAX_CUMULATIVE : INT:=10; // 最大累计不良报警数量n
MAX_CUMULATIVE_RANGE : INT:=999; // 最大累计不良计算范围
MAX_ALARM : INT:=5; // 最大报警同时推送数量
MAX_BAD_NUM : INT:=30; // 最大不良类型数量

END_VAR

SetUp();

ACTION SetUp:
//---------------------------Description header 
  //================================================================================== 
  // Harmontromics / (C) Copyright (2021) 
  //----------------------------------------------------------------------------------
  // Title:               Produce
  // Comment/Function:    产量统计，OK统计，分类NG数，分类NG比例（由大到小显示）
  // Library/Family:      (that the source is dedicated to)
  // Author:              David.Wong
  // Target System: 
  // Engineering:         TIA Portal (V15.1)
  // Restrictions:        (OB types, etc.)
  // Requirements:        (hardware, technological package, etc.) 
  //----------------------------------------------------------------------------------
  // Change log table:
  // Version     | Date       | Expert in charge | Changes applied
  //-------------|------------|------------------|------------------------------------
  // 001.000.000 | 2021-12-11 | David.Wong       | First released version
  // 001.000.001 | 2022-11-8  | David.Wong       | 增加上下翻页按钮的显示/隐藏
  // 001.001.000 | 2023-3-18  | David.Wong       | 在bad内增加stationNo变量，使报警可以归属工站         
  // 001.001.001 | 2024-1-17  | Sunny.Gao        | 使用指针的方式进行寻址，lastIndex初始赋值1
  //================================================================================== 


//---------------------------SetUp -----------------------------//

	IF NOT activated THEN
		activated:=TRUE;
		vari.goodIncrements:=1;
		FOR index := 1 TO UPPER_BOUND(badVar,1) DO
			badVar[index].goodIncrements:=1;
			badVar[index].badIncrements:=1;
      badVar[index].lastIndex:=1;
		END_FOR;
	END_IF;
	//分类不良品种类数
	badTypeNum := 0;
	FOR index := 1 TO UPPER_BOUND(badVar,1)  DO
		badList[index] := 0;
		IF badVar[index].stationNo > 0 THEN
			 badVar[index].machineNo := stations[badVar[index].stationNo].machineNo;
		END_IF;
		IF badVar[index].machineNo = machine.machineNo THEN
			badTypeNum := badTypeNum + 1;
			badList[badTypeNum] := DINT_TO_INT(index);
		END_IF;
	END_FOR;
	vari.badTypeNum 	:= badTypeNum;
	vari.badList				:=badList;

	



//---------------------------General-----------------------------//
  
  //数据清零
  clearTimer(IN := vari.allClearHmi,
              PT := t#1S);
  IF clearTimer.Q THEN
    vari.allClearAuto := TRUE;
  END_IF;
  IF vari.allClearAuto THEN
    vari.allClearAuto := FALSE;
    //清零前先保存历史数据
    IF data.totalValue > 0 THEN
      lastProduce.totalValue := data.totalValue;
      lastProduce.goodValue := data.goodValue;
      lastProduce.badValue := data.badValue;
      lastProduce.yieldRatio := data.yieldRatio;
      lastProduce.badRatio := data.badRatio;
    END_IF;
    //清零机器产量数据
    data.totalValue := 0;
    data.goodValue := 0;
    data.badValue := 0;
    data.yieldRatio := 0.0;
    data.badRatio := 0.0;
    //清零归属机器的所有不良品数据
    FOR index := 0 TO badTypeNum DO
      No := badList[index];
      badVar[No].empty := TRUE;
    END_FOR;
  END_IF;

//---------------------------Good Statistic-----------------------------//
  
  IF NOT goodExecuteCache[0] AND vari.goodExecute THEN
    data.goodValue := data.goodValue + vari.goodIncrements;
    data.cumulativeValue := data.cumulativeValue + vari.goodIncrements;
  END_IF;
  goodExecuteCache[0] := vari.goodExecute;
  vari.goodExecute := FALSE;
  


//---------------------------Bad Statistic-----------------------------//
  
  IF badTypeNum > 0 THEN
    
    //---------------------------Count-----------------------------//
      
      FOR index := 1 TO badTypeNum DO
        
        //获取当前不良品编号
        No := badList[index];
        
        //不良报警复位并清除队列或计数
        IF NOT resetCache AND machine.reset THEN
          IF badVar[No].cumulativeAlarm THEN
            badVar[No].cumulativeAlarm := FALSE;
            badVar[No].num := 0;
            badVar[No].lastIndex := 1;
            FOR index1 := 1 TO badData[No].cumulative DO
              //badVar[No].badNumList[index1] := 0;
            numListPOINT := ADR(badVar[No].badNumList[0])+index1*SIZEOF(DINT);
            numListPOINT^ := 0;
            END_FOR;
          END_IF;
          IF badVar[No].continuousAlarm THEN
            badVar[No].continuousAlarm := FALSE;
            badVar[No].continuous := 0;
          END_IF;
        END_IF;
        
        //清空连续不良计数和不良计次列表
        IF badVar[No].empty THEN
          badVar[No].empty := FALSE;
          badData[No].quantity := 0;
          badVar[No].badRatio := 0.0;
          badVar[No].continuous := 0;
          badVar[No].num := 0;
          badVar[No].lastIndex := 1;
          FOR index1 := 0 TO MAX_CUMULATIVE DO
            //badVar[No].badNumList[index1] := 0;
            numListPOINT := ADR(badVar[No].badNumList[0])+index1*SIZEOF(DINT);
            numListPOINT^ := 0;
          END_FOR;
        END_IF;
        
        //分类不良触发计数
        IF NOT badExecuteCache[No] AND badVar[No].badExecute THEN//不良品计数
          badData[No].quantity := badData[No].quantity + badVar[No].badIncrements;
          data.cumulativeValue := data.cumulativeValue + badVar[No].badIncrements;
          //累计不良计数
          IF badData[No].cumulative > 0
            AND badData[No].cumulative <= badData[No].cumulativeRange
          THEN
            //不良增量数是多少就循环多少次
            FOR index1 := 1 TO MAX( badVar[No].badIncrements, 1) DO
              badVar[No].num := badVar[No].num + 1;
              //badVar[No].badNumList[badVar[No].lastIndex] := badVar[No].num;
              numListPOINT := ADR(badVar[No].badNumList[0])+badVar[No].lastIndex*SIZEOF(DINT);
              numListPOINT^ := badVar[No].num;
              //数组索引达到最大值后从1开始
              IF badVar[No].lastIndex < badData[No].cumulative THEN
                badVar[No].lastIndex := badVar[No].lastIndex + 1;
              ELSE
                badVar[No].lastIndex := 1;
              END_IF;
            END_FOR;
            //获取不良计数最大和最小值
            maxValue := 0;
            minValue := 2147483647;
            FOR index1 := 1 TO badData[No].cumulative DO
              numListPOINT := ADR(badVar[No].badNumList[0])+index1*SIZEOF(DINT);
              IF numListPOINT^ > maxValue THEN
                maxValue := numListPOINT^;
              END_IF;
              IF numListPOINT^ < minValue THEN
                minValue := numListPOINT^;
              END_IF;        
              (*IF badVar[No].badNumList[index1] > maxValue THEN
                maxValue := badVar[No].badNumList[index1];
              END_IF;
              IF badVar[No].badNumList[index1] < minValue THEN
                minValue := badVar[No].badNumList[index1];
              END_IF;*)
            END_FOR;
            badVar[No].cumulativeAlarm := minValue > 0 AND maxValue - minValue < badData[No].cumulativeRange;
          ELSIF badVar[No].num <> 0 THEN
            //累计不良计数设置为0，清空累计不良计数
            badVar[No].num := 0;
            badVar[No].lastIndex := 1;
            FOR index1 := 0 TO MAX_CUMULATIVE DO
              badVar[No].badNumList[index1] := 0;
            END_FOR;
          END_IF;
          
          //连续不良计数
          IF badData[No].continuous > 0 THEN
            badVar[No].continuous := badVar[No].continuous + badVar[No].badIncrements;
            badVar[No].continuousAlarm := badVar[No].continuous >= badData[No].continuous;
          END_IF;
          
        ELSIF NOT goodExecuteCache[No] AND badVar[No].goodExecute THEN//良品信号
          badVar[No].continuous := 0;
          badVar[No].num := badVar[No].num + badVar[No].goodIncrements;
        END_IF;
        
        //复位计数触发
        goodExecuteCache[No] := badVar[No].goodExecute;
        badExecuteCache[No] := badVar[No].badExecute;
        badVar[No].goodExecute := FALSE;
        badVar[No].badExecute := FALSE;
        
      END_FOR;
      
    //---------------------------Bad-------------------//
              //总不良数
        totalBad := 0;
        badMax := 0;
        FOR index := 1 TO badTypeNum DO
          No := badList[index];
          totalBad :=  totalBad + badData[No].quantity;//总不良 = 分类不量[1] + 分类不量[2] + 分类不量[3] + ..........
          IF badData[No].quantity > badMax THEN
            badMax := badData[No].quantity;//分类不良中最大数
          END_IF;
        END_FOR;
        data.badValue := totalBad;
		vari.badMax 	:= totalBad;
        //总产量 = 良品产量 + 不良品产量
        data.totalValue := data.goodValue + data.badValue;
        //总良率&不良率
        IF data.totalValue > 0 THEN
          data.yieldRatio := DINT_TO_REAL(data.goodValue * 100) / DINT_TO_REAL(data.totalValue);
          data.badRatio := 100.0 - data.yieldRatio;
        ELSE
          data.yieldRatio := 0.0;
          data.badRatio := 0.0;
        END_IF;
        // 当前不良分类数量多少
        FOR index := 1 TO badTypeNum DO
          No := badList[index];
          //分类不良率方式
          IF badData[No].quantity > 0 THEN
            IF vari.percentMode = 0 AND data.totalValue > 0 THEN
              // n/总产量的分类不良率
              badVar[No].badRatio := DINT_TO_REAL(badData[No].quantity * 100) / DINT_TO_REAL(data.totalValue);
            ELSIF vari.percentMode = 1 AND data.badValue > 0 THEN
              // n/不良总数的分类不良率
              badVar[No].badRatio := DINT_TO_REAL(badData[No].quantity * 100) / DINT_TO_REAL(data.badValue);
            ELSE
              badVar[No].badRatio := 0.0;
            END_IF;
          ELSE
            badVar[No].badRatio := 0.0;
          END_IF;
        END_FOR; 
    
    //---------------------------Alarm-----------------------//      

        //获取报警状态并置位对应机器报警或工站报警，同时把报警编号存入缓存列表中
        FOR index := 1 TO badTypeNum DO
          No := badList[index];
          IF badVar[No].cumulativeAlarm OR badVar[No].continuousAlarm THEN
            IF badVar[No].stationNo > 0 THEN
              stations[badVar[No].stationNo].report.alarming := TRUE;  //置位工站报警
            ELSE
              machine.report.alarming := TRUE;  //置位机器报警
            END_IF;
          END_IF;          
        END_FOR;
    
  END_IF;
  



//---------------------------Cache 
  resetCache := machine.reset;
END_ACTION

END_FUNCTION_BLOCK

// ---- Standard/Public/06 Produce/FB_Produce_RD.TcPOU
FUNCTION_BLOCK FB_Produce_RD
VAR_IN_OUT
machine : UDT_Machine_RD; //
station : UDT_Station_RD; //
vari : UDT_ProduceVar_RD; //
data : UDT_ProduceData_RD; //
badVar : ARRAY[*] OF UDT_BadVar_RD; //
badData : ARRAY[*] OF UDT_BadData_RD; //
lastProduce : UDT_ProduceDataRecord_RD; //
END_VAR

VAR
goodExecuteCache : ARRAY[0..99] OF BOOL; // 不良触发缓存
activated : Bool; //
badExecuteCache : Array[0..99] of Bool; // 缓存不良数量
badList : Array[0..99] of Int; // 不良排序列表
maxValue : DInt; //
minValue : DInt; //
badTypeNum : Int; // 报警推送
pushAlarmNo : UInt; // 清零定时器
clearTimer : TON; // 设定定时器
resetCache : Bool; //
index : DInt; //
index1 : DInt; //
temp : DInt; //
totalBad : DInt; //
badMax : DInt; //
No : INT; //
test  : ARRAY[0..5] OF DINT;
lastIndex : DINT := 1;
index3 : INT;
numListPOINT : POINTER TO DINT;
END_VAR

VAR CONSTANT
MAX_CONTINUOUS : INT :=99; // 最大连续不良报警数量
MAX_CUMULATIVE : INT:=10; // 最大累计不良报警数量n
MAX_CUMULATIVE_RANGE : INT:=999; // 最大累计不良计算范围
MAX_ALARM : INT:=5; // 最大报警同时推送数量
MAX_BAD_NUM : INT:=30; // 最大不良类型数量

END_VAR

SetUp();
General();
GoodStatistic();
BadStatistic();
Cache();

ACTION BadStatistic:
//---------------------------Bad Statistic-----------------------------//
  
  IF badTypeNum > 0 THEN
    
    //---------------------------Count-----------------------------//
      
      FOR index := 1 TO badTypeNum DO
        
        //获取当前不良品编号
        No := badList[index];
        
        //不良报警复位并清除队列或计数
        IF NOT resetCache AND machine.reset THEN
          IF badVar[No].cumulativeAlarm THEN
            badVar[No].cumulativeAlarm := FALSE;
            badVar[No].num := 0;
            badVar[No].lastIndex := 1;
            FOR index1 := 1 TO badData[No].cumulative DO
              //badVar[No].badNumList[index1] := 0;
            numListPOINT := ADR(badVar[No].badNumList[0])+index1*SIZEOF(DINT);
            numListPOINT^ := 0;
            END_FOR;
          END_IF;
          IF badVar[No].continuousAlarm THEN
            badVar[No].continuousAlarm := FALSE;
            badVar[No].continuous := 0;
          END_IF;
        END_IF;
        
        //清空连续不良计数和不良计次列表
        IF badVar[No].empty THEN
          badVar[No].empty := FALSE;
          badData[No].quantity := 0;
          badVar[No].badRatio := 0.0;
          badVar[No].continuous := 0;
          badVar[No].num := 0;
          badVar[No].lastIndex := 1;
          FOR index1 := 0 TO MAX_CUMULATIVE DO
            //badVar[No].badNumList[index1] := 0;
            numListPOINT := ADR(badVar[No].badNumList[0])+index1*SIZEOF(DINT);
            numListPOINT^ := 0;
          END_FOR;
        END_IF;
        
        //分类不良触发计数
        IF NOT badExecuteCache[No] AND badVar[No].badExecute THEN//不良品计数
          badData[No].quantity := badData[No].quantity + badVar[No].badIncrements;
          data.cumulativeValue := data.cumulativeValue + badVar[No].badIncrements;
          //累计不良计数
          IF badData[No].cumulative > 0
            AND badData[No].cumulative <= badData[No].cumulativeRange
          THEN
            //不良增量数是多少就循环多少次
            FOR index1 := 1 TO MAX( badVar[No].badIncrements, 1) DO
              badVar[No].num := badVar[No].num + 1;
              //badVar[No].badNumList[badVar[No].lastIndex] := badVar[No].num;
              numListPOINT := ADR(badVar[No].badNumList[0])+badVar[No].lastIndex*SIZEOF(DINT);
              numListPOINT^ := badVar[No].num;
              //数组索引达到最大值后从1开始
              IF badVar[No].lastIndex < badData[No].cumulative THEN
                badVar[No].lastIndex := badVar[No].lastIndex + 1;
              ELSE
                badVar[No].lastIndex := 1;
              END_IF;
            END_FOR;
            //获取不良计数最大和最小值
            maxValue := 0;
            minValue := 2147483647;
            FOR index1 := 1 TO badData[No].cumulative DO
              numListPOINT := ADR(badVar[No].badNumList[0])+index1*SIZEOF(DINT);
              IF numListPOINT^ > maxValue THEN
                maxValue := numListPOINT^;
              END_IF;
              IF numListPOINT^ < minValue THEN
                minValue := numListPOINT^;
              END_IF;        
              (*IF badVar[No].badNumList[index1] > maxValue THEN
                maxValue := badVar[No].badNumList[index1];
              END_IF;
              IF badVar[No].badNumList[index1] < minValue THEN
                minValue := badVar[No].badNumList[index1];
              END_IF;*)
            END_FOR;
            badVar[No].cumulativeAlarm := minValue > 0 AND maxValue - minValue < badData[No].cumulativeRange;
          ELSIF badVar[No].num <> 0 THEN
            //累计不良计数设置为0，清空累计不良计数
            badVar[No].num := 0;
            badVar[No].lastIndex := 1;
            FOR index1 := 0 TO MAX_CUMULATIVE DO
              badVar[No].badNumList[index1] := 0;
            END_FOR;
          END_IF;
          
          //连续不良计数
          IF badData[No].continuous > 0 THEN
            badVar[No].continuous := badVar[No].continuous + badVar[No].badIncrements;
            badVar[No].continuousAlarm := badVar[No].continuous >= badData[No].continuous;
          END_IF;
          
        ELSIF NOT goodExecuteCache[No] AND badVar[No].goodExecute THEN//良品信号
          badVar[No].continuous := 0;
          badVar[No].num := badVar[No].num + badVar[No].goodIncrements;
        END_IF;
        
        //复位计数触发
        goodExecuteCache[No] := badVar[No].goodExecute;
        badExecuteCache[No] := badVar[No].badExecute;
        badVar[No].goodExecute := FALSE;
        badVar[No].badExecute := FALSE;
        
      END_FOR;
      
         //---------------------------Bad-------------------//
              //总不良数
        totalBad := 0;
        badMax := 0;
        FOR index := 1 TO badTypeNum DO
          No := badList[index];
          totalBad :=  totalBad + badData[No].quantity;//总不良 = 分类不量[1] + 分类不量[2] + 分类不量[3] + ..........
          IF badData[No].quantity > badMax THEN
            badMax := badData[No].quantity;//分类不良中最大数
          END_IF;
        END_FOR;
        data.badValue := totalBad;
		vari.badMax 	:= totalBad;
        //总产量 = 良品产量 + 不良品产量
        data.totalValue := data.goodValue + data.badValue;
        //总良率&不良率
        IF data.totalValue > 0 THEN
          data.yieldRatio := DINT_TO_REAL(data.goodValue * 100) / DINT_TO_REAL(data.totalValue);
          data.badRatio := 100.0 - data.yieldRatio;
        ELSE
          data.yieldRatio := 0.0;
          data.badRatio := 0.0;
        END_IF;
        // 当前不良分类数量多少
        FOR index := 1 TO badTypeNum DO
          No := badList[index];
          //分类不良率方式
          IF badData[No].quantity > 0 THEN
            IF vari.percentMode = 0 AND data.totalValue > 0 THEN
              // n/总产量的分类不良率
              badVar[No].badRatio := DINT_TO_REAL(badData[No].quantity * 100) / DINT_TO_REAL(data.totalValue);
            ELSIF vari.percentMode = 1 AND data.badValue > 0 THEN
              // n/不良总数的分类不良率
              badVar[No].badRatio := DINT_TO_REAL(badData[No].quantity * 100) / DINT_TO_REAL(data.badValue);
            ELSE
              badVar[No].badRatio := 0.0;
            END_IF;
          ELSE
            badVar[No].badRatio := 0.0;
          END_IF;
        END_FOR; 
    
    //---------------------------Alarm-----------------------//      

        //获取报警状态并置位对应机器报警或工站报警，同时把报警编号存入缓存列表中
        FOR index := 1 TO badTypeNum DO
          No := badList[index];
          IF badVar[No].cumulativeAlarm OR badVar[No].continuousAlarm THEN
            IF badVar[No].stationNo > 0 THEN
              station.report.alarming := TRUE;  //置位工站报警
            ELSE
              machine.report.alarming := TRUE;  //置位机器报警
            END_IF;
          END_IF;          
        END_FOR;
    
  END_IF;
END_ACTION

ACTION Cache:
//---------------------------Cache 
  resetCache := machine.reset;
END_ACTION

ACTION General:
//---------------------------General-----------------------------//
  
  //数据清零
  clearTimer(IN := vari.allClearHmi,
              PT := t#1S);
  IF clearTimer.Q THEN
    vari.allClearAuto := TRUE;
  END_IF;
  IF vari.allClearAuto THEN
    vari.allClearAuto := FALSE;
    //清零前先保存历史数据
    IF data.totalValue > 0 THEN
      lastProduce.totalValue := data.totalValue;
      lastProduce.goodValue := data.goodValue;
      lastProduce.badValue := data.badValue;
      lastProduce.yieldRatio := data.yieldRatio;
      lastProduce.badRatio := data.badRatio;
    END_IF;
    //清零机器产量数据
    data.totalValue := 0;
    data.goodValue := 0;
    data.badValue := 0;
    data.yieldRatio := 0.0;
    data.badRatio := 0.0;
    //清零归属机器的所有不良品数据
    FOR index := 0 TO badTypeNum DO
      No := badList[index];
      badVar[No].empty := TRUE;
    END_FOR;
  END_IF;
END_ACTION

ACTION GoodStatistic:
//---------------------------Good Statistic-----------------------------//
  
  IF NOT goodExecuteCache[0] AND vari.goodExecute THEN
    data.goodValue := data.goodValue + vari.goodIncrements;
    data.cumulativeValue := data.cumulativeValue + vari.goodIncrements;
  END_IF;
  goodExecuteCache[0] := vari.goodExecute;
  vari.goodExecute := FALSE;
END_ACTION

ACTION SetUp:
//---------------------------Description header 
  //================================================================================== 
  // Harmontromics / (C) Copyright (2021) 
  //----------------------------------------------------------------------------------
  // Title:               Produce
  // Comment/Function:    产量统计，OK统计，分类NG数，分类NG比例（由大到小显示）
  // Library/Family:      (that the source is dedicated to)
  // Author:              David.Wong
  // Target System: 
  // Engineering:         TIA Portal (V15.1)
  // Restrictions:        (OB types, etc.)
  // Requirements:        (hardware, technological package, etc.) 
  //----------------------------------------------------------------------------------
  // Change log table:
  // Version     | Date       | Expert in charge | Changes applied
  //-------------|------------|------------------|------------------------------------
  // 001.000.000 | 2021-12-11 | David.Wong       | First released version
  // 001.000.001 | 2022-11-8  | David.Wong       | 增加上下翻页按钮的显示/隐藏
  // 001.001.000 | 2023-3-18  | David.Wong       | 在bad内增加stationNo变量，使报警可以归属工站         
  // 001.001.001 | 2024-1-17  | Sunny.Gao        | 使用指针的方式进行寻址，lastIndex初始赋值1
  //================================================================================== 


//---------------------------SetUp -----------------------------//

	IF NOT activated THEN
		activated:=TRUE;
		vari.goodIncrements:=1;
		FOR index := 1 TO UPPER_BOUND(badVar,1) DO
			badVar[index].goodIncrements:=1;
			badVar[index].badIncrements:=1;
      badVar[index].lastIndex:=1;
		END_FOR;
	END_IF;
	//分类不良品种类数
	badTypeNum := 0;
	FOR index := 1 TO UPPER_BOUND(badVar,1)  DO
		badList[index] := 0;
		//IF badVar[index].stationNo > 0 THEN
		//	 badVar[index].machineNo := stations[badVar[index].stationNo].machineNo;
		//END_IF;
		IF badVar[index].machineNo = machine.machineNo THEN
			badTypeNum := badTypeNum + 1;
			badList[badTypeNum] := DINT_TO_INT(index);
		END_IF;
	END_FOR;
	vari.badTypeNum 	:= badTypeNum;
	vari.badList				:=badList;
END_ACTION

END_FUNCTION_BLOCK

// ---- Standard/FUN/FUN_AryToWord_RD.TcPOU
FUNCTION FUN_AryToWord_RD : WORD
VAR_IN_OUT
 IN : ARRAY[*] OF BOOL;
END_VAR
VAR
    index : INT;
END_VAR

FUN_AryToWord_RD.0 := IN[0];
FUN_AryToWord_RD.1 := IN[1];
FUN_AryToWord_RD.2 := IN[2];
FUN_AryToWord_RD.3 := IN[3];
FUN_AryToWord_RD.4 := IN[4];
FUN_AryToWord_RD.5 := IN[5];
FUN_AryToWord_RD.6 := IN[6];
FUN_AryToWord_RD.7 := IN[7];
FUN_AryToWord_RD.8 := IN[8];
FUN_AryToWord_RD.9 := IN[9];
FUN_AryToWord_RD.10 := IN[10];
FUN_AryToWord_RD.11 := IN[11];
FUN_AryToWord_RD.12 := IN[12];
FUN_AryToWord_RD.13 := IN[13];
FUN_AryToWord_RD.14 := IN[14];
FUN_AryToWord_RD.15 := IN[15];

END_FUNCTION

// ---- Standard/FUN/FUN_AryToLword_RD.TcPOU
FUNCTION FUN_AryToLword_RD : LWORD
VAR_IN_OUT
 IN : ARRAY[*] OF BOOL;
END_VAR
VAR
    index : INT;
END_VAR

FUN_AryToLword_RD.0 := IN[0];
FUN_AryToLword_RD.1 := IN[1];
FUN_AryToLword_RD.2 := IN[2];
FUN_AryToLword_RD.3 := IN[3];
FUN_AryToLword_RD.4 := IN[4];
FUN_AryToLword_RD.5 := IN[5];
FUN_AryToLword_RD.6 := IN[6];
FUN_AryToLword_RD.7 := IN[7];
FUN_AryToLword_RD.8 := IN[8];
FUN_AryToLword_RD.9 := IN[9];
FUN_AryToLword_RD.10 := IN[10];
FUN_AryToLword_RD.11 := IN[11];
FUN_AryToLword_RD.12 := IN[12];
FUN_AryToLword_RD.13 := IN[13];
FUN_AryToLword_RD.14 := IN[14];
FUN_AryToLword_RD.15 := IN[15];
FUN_AryToLword_RD.16 := IN[16];
FUN_AryToLword_RD.17 := IN[17];
FUN_AryToLword_RD.18 := IN[18];
FUN_AryToLword_RD.19 := IN[19];
FUN_AryToLword_RD.20 := IN[20];
FUN_AryToLword_RD.21 := IN[21];
FUN_AryToLword_RD.22 := IN[22];
FUN_AryToLword_RD.23 := IN[23];
FUN_AryToLword_RD.24 := IN[24];
FUN_AryToLword_RD.25 := IN[25];
FUN_AryToLword_RD.26 := IN[26];
FUN_AryToLword_RD.27 := IN[27];
FUN_AryToLword_RD.28 := IN[28];
FUN_AryToLword_RD.29 := IN[29];
FUN_AryToLword_RD.30 := IN[30];
FUN_AryToLword_RD.31 := IN[31];
FUN_AryToLword_RD.32 := IN[32];
FUN_AryToLword_RD.33 := IN[33];
FUN_AryToLword_RD.34 := IN[34];
FUN_AryToLword_RD.35 := IN[35];
FUN_AryToLword_RD.36 := IN[36];
FUN_AryToLword_RD.37 := IN[37];
FUN_AryToLword_RD.38 := IN[38];
FUN_AryToLword_RD.39 := IN[39];
FUN_AryToLword_RD.40 := IN[40];
FUN_AryToLword_RD.41 := IN[41];
FUN_AryToLword_RD.42 := IN[42];
FUN_AryToLword_RD.43 := IN[43];
FUN_AryToLword_RD.44 := IN[44];
FUN_AryToLword_RD.45 := IN[45];
FUN_AryToLword_RD.46 := IN[46];
FUN_AryToLword_RD.47 := IN[47];
FUN_AryToLword_RD.48 := IN[48];
FUN_AryToLword_RD.49 := IN[49];
FUN_AryToLword_RD.50 := IN[50];
FUN_AryToLword_RD.51 := IN[51];
FUN_AryToLword_RD.52 := IN[52];
FUN_AryToLword_RD.53 := IN[53];
FUN_AryToLword_RD.54 := IN[54];
FUN_AryToLword_RD.55 := IN[55];
FUN_AryToLword_RD.56 := IN[56];
FUN_AryToLword_RD.57 := IN[57];
FUN_AryToLword_RD.58 := IN[58];
FUN_AryToLword_RD.59 := IN[59];
FUN_AryToLword_RD.60 := IN[60];
FUN_AryToLword_RD.61 := IN[61];
FUN_AryToLword_RD.62 := IN[62];
FUN_AryToLword_RD.63 := IN[63];

END_FUNCTION

// ---- Standard/Module/FAKRA/BraidFlaring/FB_BraidFlaring_RD.TcPOU
FUNCTION_BLOCK FB_BraidFlaring_RD

VAR_IN_OUT
  BraidFlaring : UDT_BraidFlaring_RD;
  BraidFlaringData : UDT_Data_BraidFlaring_RD;
END_VAR

VAR_INPUT
	//BraidFlaring 模组接口
  HomeSensor_gripCyl : BOOL;
  WorkSensor_gripCyl : BOOL;
  HomeValve_gripCyl : BOOL;
  WorkValve_gripCyl : BOOL;
  HomeLabel_gripCyl : STRING[10];
  WorkLabel_gripCyl : STRING[10];
   
  HomeSensor_jackCyl : BOOL;
  WorkSensor_jackCyl : BOOL;
  HomeValve_jackCyl : BOOL;
  WorkValve_jackCyl : BOOL;
  HomeLabel_jackCyl : STRING[10];
  WorkLabel_jackCyl : STRING[10];
  
  HomeSensor_pushCyl : BOOL;
  WorkSensor_pushCyl : BOOL;
  HomeValve_pushCyl : BOOL;
  WorkValve_pushCyl : BOOL;
  HomeLabel_pushCyl : STRING[10];
  WorkLabel_pushCyl : STRING[10];
  
  HomeValve_blow    : BOOL;
  WorkValve_blow    : BOOL;
  
  HomeValve_vacuum  : BOOL;
  WorkValve_vacuum  : BOOL;
  
  pushRodInPos      : BOOL;
  
  //GS 传送线接口
  HomeSensor_fixCyl : BOOL;
  WorkSensor_fixCyl : BOOL;
  HomeValve_fixCyl : BOOL;
  WorkValve_fixCyl : BOOL;
  HomeLabel_fixCyl : STRING[10];
  WorkLabel_fixCyl : STRING[10];
  
  HomeSensor_stepFixCyl : BOOL;
  WorkSensor_stepFixCyl : BOOL;
  HomeValve_stepFixCyl : BOOL;
  WorkValve_stepFixCyl : BOOL;
  HomeLabel_stepFixCyl : STRING[10];
  WorkLabel_stepFixCyl : STRING[10];
END_VAR

VAR  
  machine      		: UDT_Machine_RD;
  station      		: UDT_Station_RD;
  
  gripCyl	   		:UDT_CylinderVar_RD;
  jackCyl   		:UDT_CylinderVar_RD;
  pushCyl   		:UDT_CylinderVar_RD;
  fixCyl       		:UDT_CylinderVar_RD;
  stepFixCyl    	:UDT_CylinderVar_RD; 
  blow              :UDT_CylinderVar_RD;
  vacuum            :UDT_CylinderVar_RD;
  
  transferAxis 		: UDT_AxisVar_RD; 
  rotateAxis 		: UDT_AxisVar_RD;  
  
 
  fB_BraidFlaring		: FB_Station_RD;
  fB_gripCyl			: FB_Cylinder_RD;
  fB_jackCyl			: FB_Cylinder_RD;
  fB_pushCyl			: FB_Cylinder_RD;
  fB_fixCyl         	: FB_Cylinder_RD;  
  fB_stepFixCyl     	: FB_Cylinder_RD; 
  fB_blow               : FB_Cylinder_RD;
  fB_vacuum             : FB_Cylinder_RD;
  
  fb_transferAxis		: FB_Axis_RD;
  fb_rotateAxis			: FB_Axis_RD;
  
  activated             : BOOL;
  
  tonPushRodNotInPos    : TON;
  pushRodNotInPos       : BOOL;
  
  RunningExcept         : BOOL;  //运行中除外
  
END_VAR

VAR CONSTANT
  INIT :INT := 0;
  AUTO :INT := 1;
  AUTO2 :INT :=2;
  
  //TransferAxis
  HOME_TRANS              : UINT:=1;
  FIRST_CLIP_TRANS        : UINT:=2;
  SECOND_CLIP_TRANS		  : UINT:=3;
  THIRD_CLIP_TRANS		  : UINT:=4;
  PUSH_STRAT_TRANS        : UINT:=5;
  PUSH_END_TRANS          : UINT:=6;
//  CLIP_TRANS              : UINT:=7;
  
    //rotateAxis
  HOME_ROTATE             : UINT:=1;
  FIRST_CLIP_ROTATE       : UINT:=2;
  SECOND_CLIP_ROTATE      : UINT:=3;
  THIRD_CLIP_ROTATE 	  : UINT:=4;
  PUSH_ROTATE             : UINT:=5; 
//  CLIP_ROTATE             : UINT:=6; 

END_VAR

SetUp();
Command();
General();
Permit();
StepInit();
StepAuto();
Alarm();
AutoTip();
ManualTip();
Tip();
Hmi();

ACTION Alarm:
BraidFlaring.Message.userAlarms[0] := gripCyl.homeSensorOffAlarm[0];
BraidFlaring.Message.userAlarms[1] := gripCyl.homeSensorOnAlarm[0];
BraidFlaring.Message.userAlarms[2] := gripCyl.workSensorOffAlarm[0];
BraidFlaring.Message.userAlarms[3] := gripCyl.workSensorOnAlarm[0];

BraidFlaring.Message.userAlarms[4] := jackCyl.homeSensorOffAlarm[0];
BraidFlaring.Message.userAlarms[5] := jackCyl.homeSensorOnAlarm[0];
BraidFlaring.Message.userAlarms[6] := jackCyl.workSensorOffAlarm[0];
BraidFlaring.Message.userAlarms[7] := jackCyl.workSensorOnAlarm[0];

BraidFlaring.Message.userAlarms[8] := pushCyl.homeSensorOffAlarm[0];
BraidFlaring.Message.userAlarms[9] := pushCyl.homeSensorOnAlarm[0];
BraidFlaring.Message.userAlarms[10] := pushCyl.workSensorOffAlarm[0];
BraidFlaring.Message.userAlarms[11] := pushCyl.workSensorOnAlarm[0];

BraidFlaring.Message.userAlarms[12] := fixCyl.homeSensorOffAlarm[0];
BraidFlaring.Message.userAlarms[13] := fixCyl.homeSensorOnAlarm[0];
BraidFlaring.Message.userAlarms[14] := fixCyl.workSensorOffAlarm[0];
BraidFlaring.Message.userAlarms[15] := fixCyl.workSensorOnAlarm[0];

BraidFlaring.Message.userAlarms[16] := stepFixCyl.homeSensorOffAlarm[0];
BraidFlaring.Message.userAlarms[17] := stepFixCyl.homeSensorOnAlarm[0];
BraidFlaring.Message.userAlarms[18] := stepFixCyl.workSensorOffAlarm[0];
BraidFlaring.Message.userAlarms[19] := stepFixCyl.workSensorOnAlarm[0];

BraidFlaring.Message.userAlarms[20] := transferAxis.alarming;
BraidFlaring.Message.userAlarms[21] := rotateAxis.alarming;

tonPushRodNotInPos(IN:=NOT pushRodInPos,PT:=T#1S,Q=>,ET=>);
IF tonPushRodNotInPos.Q THEN
	pushRodNotInPos:=TRUE;
END_IF


BraidFlaring.Message.presetAlarms[0] :=station.presetAlarms[0];//工站初始化超时报警

IF machine.reset
THEN
	pushRodNotInPos:=FALSE;
END_IF
END_ACTION

ACTION AutoTip:
BraidFlaring.Message.userAutoTips[0] := gripCyl.autoTip ;
BraidFlaring.Message.userAutoTips[1] := jackCyl.autoTip ;
BraidFlaring.Message.userAutoTips[2] := pushCyl.autoTip ;
BraidFlaring.Message.userAutoTips[3] := fixCyl.autoTip ;
BraidFlaring.Message.userAutoTips[4] := stepFixCyl.autoTip ;

